LIN {X 0,Y 198.265,Z 302.232,A -85,B 0,C 180,E1 -25531.624,E2 -25531.624} C_VEL
LIN {X 0,Y 201.477,Z 266.48,A -85,B 0,C 180,E1 -25532.577,E2 -25532.577} C_VEL
LIN {X 0,Y 197.128,Z 257.364,A -85,B 0,C 180,E1 -25535.935,E2 -25535.935} C_VEL
LIN {X 0,Y 193.487,Z 250.577,A -85,B 0,C 180,E1 -25539.188,E2 -25539.188} C_VEL
LIN {X 0,Y 190.353,Z 244.979,A -85,B 0,C 180,E1 -25542.543,E2 -25542.543} C_VEL
LIN {X 0,Y 187.689,Z 240.639,A -85,B 0,C 180,E1 -25546.051,E2 -25546.051} C_VEL
LIN {X 0,Y 185.533,Z 236.807,A -85,B 0,C 180,E1 -25549.91,E2 -25549.91} C_VEL
LIN {X 0,Y 183.726,Z 233.495,A -85,B 0,C 180,E1 -25555.359,E2 -25555.359} C_VEL
LIN {X 0,Y 183.496,Z 232.327,A -85,B 0,C 180,E1 -25557.256,E2 -25557.256} C_VEL
LIN {X 0,Y 183.478,Z 232.249,A -85,B 0,C 180,E1 -25562.195,E2 -25562.195} C_VEL
LIN {X 0,Y 183.641,Z 233.069,A -85,B 0,C 180,E1 -25563.703,E2 -25563.703} C_VEL
LIN {X 0,Y 185.447,Z 236.708,A -85,B 0,C 180,E1 -25569.566,E2 -25569.566} C_VEL
LIN {X 0,Y 186.036,Z 237.651,A -85,B 0,C 180,E1 -25570.761,E2 -25570.761} C_VEL
LIN {X 0,Y 188.522,Z 241.906,A -85,B 0,C 180,E1 -25574.781,E2 -25574.781} C_VEL
LIN {X 0,Y 190.791,Z 245.771,A -85,B 0,C 180,E1 -25577.622,E2 -25577.622} C_VEL
LIN {X 0,Y 194.145,Z 251.69,A -85,B 0,C 180,E1 -25581.084,E2 -25581.084} C_VEL
LIN {X 0,Y 196.253,Z 256.423,A -85,B 0,C 180,E1 -25583.047,E2 -25583.047} C_VEL
LIN {X 0,Y 199.614,Z 265.237,A -85,B 0,C 180,E1 -25585.917,E2 -25585.917} C_VEL
LIN {X 0,Y 201.248,Z 269.943,A -85,B 0,C 180,E1 -25587.212,E2 -25587.212} C_VEL
LIN {X 0,Y 196.172,Z 324.072,A -85,B 0,C 180,E1 -25588.661,E2 -25588.661} C_VEL
LIN {X 0,Y 193.425,Z 339.856,A -85,B 0,C 180,E1 -25589.304,E2 -25589.304} C_VEL
LIN {X 0,Y 189.575,Z 355.078,A -85,B 0,C 180,E1 -25590.202,E2 -25590.202} C_VEL
LIN {X 0,Y 185.022,Z 368.797,A -85,B 0,C 180,E1 -25591.278,E2 -25591.278} C_VEL
LIN {X 0,Y 179.622,Z 382.244,A -85,B 0,C 180,E1 -25592.73,E2 -25592.73} C_VEL
LIN {X 0,Y 173.751,Z 394.633,A -85,B 0,C 180,E1 -25594.491,E2 -25594.491} C_VEL
LIN {X 0,Y 166.772,Z 407.28,A -85,B 0,C 180,E1 -25596.804,E2 -25596.804} C_VEL
LIN {X 0,Y 159.475,Z 418.758,A -85,B 0,C 180,E1 -25599.536,E2 -25599.536} C_VEL
LIN {X 0,Y 152.63,Z 428.424,A -85,B 0,C 180,E1 -25602.545,E2 -25602.545} C_VEL
LIN {X 0,Y 146.12,Z 436.937,A -85,B 0,C 180,E1 -25605.972,E2 -25605.972} C_VEL
LIN {X 0,Y 139.146,Z 445.515,A -85,B 0,C 180,E1 -25610.535,E2 -25610.535} C_VEL
LIN {X 0,Y 132.201,Z 453.257,A -85,B 0,C 180,E1 -25616.069,E2 -25616.069} C_VEL
LIN {X 0,Y 127.367,Z 458.659,A -85,B 0,C 180,E1 -25621.381,E2 -25621.381} C_VEL
LIN {X 0,Y 125.007,Z 460.662,A -85,B 0,C 180,E1 -25623.675,E2 -25623.675} C_VEL
LIN {X 0,Y 119.764,Z 463.476,A -85,B 0,C 180,E1 -25627.4,E2 -25627.4} C_VEL
LIN {X 0,Y 115.776,Z 465.338,A -85,B 0,C 180,E1 -25630.633,E2 -25630.633} C_VEL
LIN {X 0,Y 113.774,Z 466.531,A -85,B 0,C 180,E1 -25633.354,E2 -25633.354} C_VEL
LIN {X 0,Y 113.422,Z 466.832,A -85,B 0,C 180,E1 -25634.315,E2 -25634.315} C_VEL
LIN {X 0,Y 112.458,Z 468.336,A -85,B 0,C 180,E1 -25639.194,E2 -25639.194} C_VEL
LIN {X 0,Y 112.095,Z 469.523,A -85,B 0,C 180,E1 -25646.405,E2 -25646.405} C_VEL
LIN {X 0,Y 112.248,Z 469.683,A -85,B 0,C 180,E1 -25650,E2 -25650} C_VEL
LIN {X 0,Y 112.127,Z 469.052,A -85,B 0,C 180,E1 -25657.201,E2 -25657.201} C_VEL
LIN {X 0,Y 113.102,Z 467.265,A -85,B 0,C 180,E1 -25664.392,E2 -25664.392} C_VEL
LIN {X 0,Y 115.542,Z 464.307,A -85,B 0,C 180,E1 -25671.405,E2 -25671.405} C_VEL
LIN {X 0,Y 119.379,Z 460.108,A -85,B 0,C 180,E1 -25678.097,E2 -25678.097} C_VEL
LIN {X 0,Y 124.74,Z 454.565,A -85,B 0,C 180,E1 -25684.292,E2 -25684.292} C_VEL
LIN {X 0,Y 131.461,Z 447.53,A -85,B 0,C 180,E1 -25689.906,E2 -25689.906} C_VEL
LIN {X 0,Y 138.147,Z 439.961,A -85,B 0,C 180,E1 -25694.428,E2 -25694.428} C_VEL
LIN {X 0,Y 145.577,Z 430.948,A -85,B 0,C 180,E1 -25698.443,E2 -25698.443} C_VEL
LIN {X 0,Y 153.784,Z 420.066,A -85,B 0,C 180,E1 -25702.03,E2 -25702.03} C_VEL
LIN {X 0,Y 161.304,Z 408.87,A -85,B 0,C 180,E1 -25704.78,E2 -25704.78} C_VEL
LIN {X 0,Y 168.57,Z 396.421,A -85,B 0,C 180,E1 -25707.123,E2 -25707.123} C_VEL
LIN {X 0,Y 175.175,Z 383.102,A -85,B 0,C 180,E1 -25709.044,E2 -25709.044} C_VEL
LIN {X 0,Y 180.736,Z 369.84,A -85,B 0,C 180,E1 -25710.466,E2 -25710.466} C_VEL
LIN {X 0,Y 185.351,Z 356.452,A -85,B 0,C 180,E1 -25711.547,E2 -25711.547} C_VEL
LIN {X 0,Y 189.311,Z 341.786,A -85,B 0,C 180,E1 -25712.417,E2 -25712.417} C_VEL
LIN {X 0,Y 192.254,Z 326.282,A -85,B 0,C 180,E1 -25713.068,E2 -25713.068} C_VEL
LIN {X 0,Y 194.747,Z 303.203,A -85,B 0,C 180,E1 -25713.707,E2 -25713.707} C_VEL
LIN {X 0,Y 197.576,Z 272.684,A -85,B 0,C 180,E1 -25714.507,E2 -25714.507} C_VEL
LIN {X 0,Y 194.287,Z 263.272,A -85,B 0,C 180,E1 -25717.468,E2 -25717.468} C_VEL
LIN {X 0,Y 192.199,Z 258.069,A -85,B 0,C 180,E1 -25719.533,E2 -25719.533} C_VEL
LIN {X 0,Y 189.081,Z 252.283,A -85,B 0,C 180,E1 -25722.91,E2 -25722.91} C_VEL
LIN {X 0,Y 186.331,Z 247.346,A -85,B 0,C 180,E1 -25726.643,E2 -25726.643} C_VEL
LIN {X 0,Y 184.285,Z 243.616,A -85,B 0,C 180,E1 -25730.396,E2 -25730.396} C_VEL
LIN {X 0,Y 182.602,Z 240.468,A -85,B 0,C 180,E1 -25735.447,E2 -25735.447} C_VEL
LIN {X 0,Y 182.361,Z 239.282,A -85,B 0,C 180,E1 -25737.239,E2 -25737.239} C_VEL
LIN {X 0,Y 182.233,Z 239.216,A -85,B 0,C 180,E1 -25742.21,E2 -25742.21} C_VEL
LIN {X 0,Y 182.442,Z 239.623,A -85,B 0,C 180,E1 -25743.866,E2 -25743.866} C_VEL
LIN {X 0,Y 183.716,Z 242.998,A -85,B 0,C 180,E1 -25748.802,E2 -25748.802} C_VEL
LIN {X 0,Y 184.522,Z 244.089,A -85,B 0,C 180,E1 -25750.562,E2 -25750.562} C_VEL
LIN {X 0,Y 186.922,Z 248.505,A -85,B 0,C 180,E1 -25754.702,E2 -25754.702} C_VEL
LIN {X 0,Y 189.301,Z 252.766,A -85,B 0,C 180,E1 -25757.8,E2 -25757.8} C_VEL
LIN {X 0,Y 192.242,Z 258.192,A -85,B 0,C 180,E1 -25760.952,E2 -25760.952} C_VEL
LIN {X 0,Y 195.843,Z 265.523,A -85,B 0,C 180,E1 -25764.233,E2 -25764.233} C_VEL
LIN {X 0,Y 197.757,Z 269.776,A -85,B 0,C 180,E1 -25765.802,E2 -25765.802} C_VEL
LIN {X 0,Y 193.116,Z 318.432,A -85,B 0,C 180,E1 -25767.116,E2 -25767.116} C_VEL
LIN {X 0,Y 190.335,Z 334.317,A -85,B 0,C 180,E1 -25767.744,E2 -25767.744} C_VEL
LIN {X 0,Y 186.373,Z 350.163,A -85,B 0,C 180,E1 -25768.748,E2 -25768.748} C_VEL
LIN {X 0,Y 181.609,Z 364.66,A -85,B 0,C 180,E1 -25770.016,E2 -25770.016} C_VEL
LIN {X 0,Y 176.331,Z 377.734,A -85,B 0,C 180,E1 -25771.522,E2 -25771.522} C_VEL
LIN {X 0,Y 169.714,Z 391.314,A -85,B 0,C 180,E1 -25773.551,E2 -25773.551} C_VEL
LIN {X 0,Y 162.629,Z 403.514,A -85,B 0,C 180,E1 -25775.877,E2 -25775.877} C_VEL
LIN {X 0,Y 155.241,Z 414.63,A -85,B 0,C 180,E1 -25778.654,E2 -25778.654} C_VEL
LIN {X 0,Y 148.173,Z 424.142,A -85,B 0,C 180,E1 -25781.784,E2 -25781.784} C_VEL
LIN {X 0,Y 141.937,Z 431.925,A -85,B 0,C 180,E1 -25785.123,E2 -25785.123} C_VEL
LIN {X 0,Y 134.944,Z 439.778,A -85,B 0,C 180,E1 -25789.382,E2 -25789.382} C_VEL
LIN {X 0,Y 127.923,Z 447.104,A -85,B 0,C 180,E1 -25794.77,E2 -25794.77} C_VEL
LIN {X 0,Y 122.164,Z 452.906,A -85,B 0,C 180,E1 -25800.725,E2 -25800.725} C_VEL
LIN {X 0,Y 118.72,Z 456.337,A -85,B 0,C 180,E1 -25805.519,E2 -25805.519} C_VEL
LIN {X 0,Y 115.274,Z 459.803,A -85,B 0,C 180,E1 -25812.252,E2 -25812.252} C_VEL
LIN {X 0,Y 113.203,Z 462.086,A -85,B 0,C 180,E1 -25819.266,E2 -25819.266} C_VEL
LIN {X 0,Y 112.353,Z 463.242,A -85,B 0,C 180,E1 -25826.414,E2 -25826.414} C_VEL
LIN {X 0,Y 112.335,Z 463.394,A -85,B 0,C 180,E1 -25830,E2 -25830} C_VEL
LIN {X 0,Y 112.624,Z 462.835,A -85,B 0,C 180,E1 -25837.17,E2 -25837.17} C_VEL
LIN {X 0,Y 114.052,Z 461.162,A -85,B 0,C 180,E1 -25844.27,E2 -25844.27} C_VEL
LIN {X 0,Y 116.719,Z 458.337,A -85,B 0,C 180,E1 -25851.179,E2 -25851.179} C_VEL
LIN {X 0,Y 120.935,Z 454.278,A -85,B 0,C 180,E1 -25857.705,E2 -25857.705} C_VEL
LIN {X 0,Y 126.325,Z 448.897,A -85,B 0,C 180,E1 -25863.804,E2 -25863.804} C_VEL
LIN {X 0,Y 133.008,Z 442.029,A -85,B 0,C 180,E1 -25869.351,E2 -25869.351} C_VEL
LIN {X 0,Y 140.793,Z 433.449,A -85,B 0,C 180,E1 -25874.335,E2 -25874.335} C_VEL
LIN {X 0,Y 148.026,Z 424.662,A -85,B 0,C 180,E1 -25878.165,E2 -25878.165} C_VEL
LIN {X 0,Y 155.16,Z 415.03,A -85,B 0,C 180,E1 -25881.384,E2 -25881.384} C_VEL
LIN {X 0,Y 163.16,Z 402.982,A -85,B 0,C 180,E1 -25884.393,E2 -25884.393} C_VEL
LIN {X 0,Y 170.261,Z 390.675,A -85,B 0,C 180,E1 -25886.707,E2 -25886.707} C_VEL
LIN {X 0,Y 176.412,Z 378.03,A -85,B 0,C 180,E1 -25888.585,E2 -25888.585} C_VEL
LIN {X 0,Y 181.47,Z 365.506,A -85,B 0,C 180,E1 -25890.06,E2 -25890.06} C_VEL
LIN {X 0,Y 186.272,Z 351.22,A -85,B 0,C 180,E1 -25891.309,E2 -25891.309} C_VEL
LIN {X 0,Y 190.119,Z 336.499,A -85,B 0,C 180,E1 -25892.238,E2 -25892.238} C_VEL
LIN {X 0,Y 192.878,Z 321.586,A -85,B 0,C 180,E1 -25892.902,E2 -25892.902} C_VEL
LIN {X 0,Y 195.246,Z 299.869,A -85,B 0,C 180,E1 -25893.515,E2 -25893.515} C_VEL
LIN {X 0,Y 198.046,Z 270.082,A -85,B 0,C 180,E1 -25894.274,E2 -25894.274} C_VEL
LIN {X 0,Y 194.366,Z 262.13,A -85,B 0,C 180,E1 -25897.389,E2 -25897.389} C_VEL
LIN {X 0,Y 190.853,Z 255.339,A -85,B 0,C 180,E1 -25900.854,E2 -25900.854} C_VEL
LIN {X 0,Y 188.192,Z 250.581,A -85,B 0,C 180,E1 -25904.013,E2 -25904.013} C_VEL
LIN {X 0,Y 186.382,Z 247.347,A -85,B 0,C 180,E1 -25906.639,E2 -25906.639} C_VEL
LIN {X 0,Y 184.409,Z 243.664,A -85,B 0,C 180,E1 -25910.402,E2 -25910.402} C_VEL
LIN {X 0,Y 182.727,Z 240.167,A -85,B 0,C 180,E1 -25916.14,E2 -25916.14} C_VEL
LIN {X 0,Y 182.572,Z 239.291,A -85,B 0,C 180,E1 -25917.794,E2 -25917.794} C_VEL
LIN {X 0,Y 182.613,Z 239.299,A -85,B 0,C 180,E1 -25922.205,E2 -25922.205} C_VEL
LIN {X 0,Y 184.443,Z 243.691,A -85,B 0,C 180,E1 -25929.319,E2 -25929.319} C_VEL
LIN {X 0,Y 187.034,Z 248.381,A -85,B 0,C 180,E1 -25933.998,E2 -25933.998} C_VEL
LIN {X 0,Y 189.551,Z 252.95,A -85,B 0,C 180,E1 -25937.324,E2 -25937.324} C_VEL
LIN {X 0,Y 192.628,Z 258.726,A -85,B 0,C 180,E1 -25940.628,E2 -25940.628} C_VEL
LIN {X 0,Y 195.09,Z 265.052,A -85,B 0,C 180,E1 -25943.041,E2 -25943.041} C_VEL
LIN {X 0,Y 197.801,Z 272.956,A -85,B 0,C 180,E1 -25945.465,E2 -25945.465} C_VEL
LIN {X 0,Y 192.844,Z 324.07,A -85,B 0,C 180,E1 -25946.818,E2 -25946.818} C_VEL
LIN {X 0,Y 190.047,Z 339.667,A -85,B 0,C 180,E1 -25947.435,E2 -25947.435} C_VEL
LIN {X 0,Y 186.087,Z 354.885,A -85,B 0,C 180,E1 -25948.303,E2 -25948.303} C_VEL
LIN {X 0,Y 181.436,Z 368.604,A -85,B 0,C 180,E1 -25949.361,E2 -25949.361} C_VEL
LIN {X 0,Y 175.871,Z 382.05,A -85,B 0,C 180,E1 -25950.776,E2 -25950.776} C_VEL
LIN {X 0,Y 169.385,Z 395.286,A -85,B 0,C 180,E1 -25952.642,E2 -25952.642} C_VEL
LIN {X 0,Y 161.958,Z 408.156,A -85,B 0,C 180,E1 -25955.009,E2 -25955.009} C_VEL
LIN {X 0,Y 153.809,Z 420.321,A -85,B 0,C 180,E1 -25957.982,E2 -25957.982} C_VEL
LIN {X 0,Y 145.602,Z 431.152,A -85,B 0,C 180,E1 -25961.568,E2 -25961.568} C_VEL
LIN {X 0,Y 138.413,Z 439.903,A -85,B 0,C 180,E1 -25965.472,E2 -25965.472} C_VEL
LIN {X 0,Y 131.53,Z 447.689,A -85,B 0,C 180,E1 -25970.119,E2 -25970.119} C_VEL
LIN {X 0,Y 126.304,Z 453.057,A -85,B 0,C 180,E1 -25974.249,E2 -25974.249} C_VEL
LIN {X 0,Y 120.674,Z 458.941,A -85,B 0,C 180,E1 -25980.328,E2 -25980.328} C_VEL
LIN {X 0,Y 117.361,Z 462.447,A -85,B 0,C 180,E1 -25985.217,E2 -25985.217} C_VEL
LIN {X 0,Y 114.102,Z 465.992,A -85,B 0,C 180,E1 -25992.063,E2 -25992.063} C_VEL
LIN {X 0,Y 113.422,Z 466.832,A -85,B 0,C 180,E1 -25994.315,E2 -25994.315} C_VEL
LIN {X 0,Y 112.199,Z 467.828,A -85,B 0,C 180,E1 -25997.204,E2 -25997.204} C_VEL
LIN {X 0,Y 108.998,Z 468.967,A -85,B 0,C 180,E1 -26002.012,E2 -26002.012} C_VEL
LIN {X 0,Y 105.596,Z 469.509,A -85,B 0,C 180,E1 -26008.153,E2 -26008.153} C_VEL
LIN {X 0,Y 105.135,Z 469.471,A -85,B 0,C 180,E1 -26010.309,E2 -26010.309} C_VEL
LIN {X 0,Y 105.053,Z 468.852,A -85,B 0,C 180,E1 -26017.689,E2 -26017.689} C_VEL
LIN {X 0,Y 106.184,Z 467.064,A -85,B 0,C 180,E1 -26025.352,E2 -26025.352} C_VEL
LIN {X 0,Y 108.884,Z 464.105,A -85,B 0,C 180,E1 -26032.785,E2 -26032.785} C_VEL
LIN {X 0,Y 113.108,Z 459.907,A -85,B 0,C 180,E1 -26039.807,E2 -26039.807} C_VEL
LIN {X 0,Y 118.877,Z 454.363,A -85,B 0,C 180,E1 -26046.242,E2 -26046.242} C_VEL
LIN {X 0,Y 126.045,Z 447.327,A -85,B 0,C 180,E1 -26051.997,E2 -26051.997} C_VEL
LIN {X 0,Y 133.556,Z 439.265,A -85,B 0,C 180,E1 -26056.836,E2 -26056.836} C_VEL
LIN {X 0,Y 140.943,Z 430.746,A -85,B 0,C 180,E1 -26060.615,E2 -26060.615} C_VEL
LIN {X 0,Y 149.492,Z 419.863,A -85,B 0,C 180,E1 -26064.191,E2 -26064.191} C_VEL
LIN {X 0,Y 157.306,Z 408.668,A -85,B 0,C 180,E1 -26066.898,E2 -26066.898} C_VEL
LIN {X 0,Y 165.108,Z 395.702,A -85,B 0,C 180,E1 -26069.284,E2 -26069.284} C_VEL
LIN {X 0,Y 171.628,Z 382.898,A -85,B 0,C 180,E1 -26071.079,E2 -26071.079} C_VEL
LIN {X 0,Y 177.342,Z 369.636,A -85,B 0,C 180,E1 -26072.464,E2 -26072.464} C_VEL
LIN {X 0,Y 182.076,Z 356.247,A -85,B 0,C 180,E1 -26073.512,E2 -26073.512} C_VEL
LIN {X 0,Y 186.132,Z 341.578,A -85,B 0,C 180,E1 -26074.353,E2 -26074.353} C_VEL
LIN {X 0,Y 189.091,Z 326.379,A -85,B 0,C 180,E1 -26074.978,E2 -26074.978} C_VEL
LIN {X 0,Y 191.547,Z 304.546,A -85,B 0,C 180,E1 -26075.576,E2 -26075.576} C_VEL
LIN {X 0,Y 194.298,Z 275.812,A -85,B 0,C 180,E1 -26076.313,E2 -26076.313} C_VEL
LIN {X 0,Y 191.694,Z 267.952,A -85,B 0,C 180,E1 -26078.915,E2 -26078.915} C_VEL
LIN {X 0,Y 190.099,Z 263.817,A -85,B 0,C 180,E1 -26080.636,E2 -26080.636} C_VEL
LIN {X 0,Y 186.9,Z 257.529,A -85,B 0,C 180,E1 -26084.46,E2 -26084.46} C_VEL
LIN {X 0,Y 184.856,Z 253.826,A -85,B 0,C 180,E1 -26087.512,E2 -26087.512} C_VEL
LIN {X 0,Y 183.132,Z 250.42,A -85,B 0,C 180,E1 -26090.961,E2 -26090.961} C_VEL
LIN {X 0,Y 181.628,Z 247.298,A -85,B 0,C 180,E1 -26095.979,E2 -26095.979} C_VEL
LIN {X 0,Y 181.494,Z 246.355,A -85,B 0,C 180,E1 -26097.226,E2 -26097.226} C_VEL
LIN {X 0,Y 181.279,Z 246.096,A -85,B 0,C 180,E1 -26100,E2 -26100} C_VEL
LIN {X 0,Y 181.526,Z 246.656,A -85,B 0,C 180,E1 -26103.607,E2 -26103.607} C_VEL
LIN {X 0,Y 182.764,Z 250.033,A -85,B 0,C 180,E1 -26108.639,E2 -26108.639} C_VEL
LIN {X 0,Y 183.445,Z 251.083,A -85,B 0,C 180,E1 -26110.206,E2 -26110.206} C_VEL
LIN {X 0,Y 185.533,Z 255.12,A -85,B 0,C 180,E1 -26114.029,E2 -26114.029} C_VEL
LIN {X 0,Y 187.886,Z 259.548,A -85,B 0,C 180,E1 -26117.272,E2 -26117.272} C_VEL
LIN {X 0,Y 190.91,Z 265.585,A -85,B 0,C 180,E1 -26120.664,E2 -26120.664} C_VEL
LIN {X 0,Y 193.676,Z 271.568,A -85,B 0,C 180,E1 -26123.317,E2 -26123.317} C_VEL
LIN {X 0,Y 194.461,Z 273.393,A -85,B 0,C 180,E1 -26124.018,E2 -26124.018} C_VEL
LIN {X 0,Y 189.897,Z 319.326,A -85,B 0,C 180,E1 -26125.238,E2 -26125.238} C_VEL
LIN {X 0,Y 187.147,Z 334.525,A -85,B 0,C 180,E1 -26125.828,E2 -26125.828} C_VEL
LIN {X 0,Y 183.063,Z 350.369,A -85,B 0,C 180,E1 -26126.799,E2 -26126.799} C_VEL
LIN {X 0,Y 178.165,Z 364.865,A -85,B 0,C 180,E1 -26128.04,E2 -26128.04} C_VEL
LIN {X 0,Y 172.564,Z 378.281,A -85,B 0,C 180,E1 -26129.56,E2 -26129.56} C_VEL
LIN {X 0,Y 165.9,Z 391.516,A -85,B 0,C 180,E1 -26131.509,E2 -26131.509} C_VEL
LIN {X 0,Y 158.581,Z 403.716,A -85,B 0,C 180,E1 -26133.802,E2 -26133.802} C_VEL
LIN {X 0,Y 150.896,Z 414.832,A -85,B 0,C 180,E1 -26136.542,E2 -26136.542} C_VEL
LIN {X 0,Y 143.09,Z 424.887,A -85,B 0,C 180,E1 -26139.858,E2 -26139.858} C_VEL
LIN {X 0,Y 136.996,Z 432.126,A -85,B 0,C 180,E1 -26143.027,E2 -26143.027} C_VEL
LIN {X 0,Y 129.619,Z 439.979,A -85,B 0,C 180,E1 -26147.331,E2 -26147.331} C_VEL
LIN {X 0,Y 122.176,Z 447.304,A -85,B 0,C 180,E1 -26152.843,E2 -26152.843} C_VEL
LIN {X 0,Y 115.98,Z 453.107,A -85,B 0,C 180,E1 -26158.998,E2 -26158.998} C_VEL
LIN {X 0,Y 112.283,Z 456.537,A -85,B 0,C 180,E1 -26164.015,E2 -26164.015} C_VEL
LIN {X 0,Y 108.496,Z 460.004,A -85,B 0,C 180,E1 -26171.102,E2 -26171.102} C_VEL
LIN {X 0,Y 106.216,Z 462.286,A -85,B 0,C 180,E1 -26178.551,E2 -26178.551} C_VEL
LIN {X 0,Y 105.265,Z 463.441,A -85,B 0,C 180,E1 -26186.172,E2 -26186.172} C_VEL
LIN {X 0,Y 105.237,Z 463.593,A -85,B 0,C 180,E1 -26190,E2 -26190} C_VEL
LIN {X 0,Y 105.593,Z 463.033,A -85,B 0,C 180,E1 -26197.65,E2 -26197.65} C_VEL
LIN {X 0,Y 107.158,Z 461.361,A -85,B 0,C 180,E1 -26205.209,E2 -26205.209} C_VEL
LIN {X 0,Y 110.095,Z 458.536,A -85,B 0,C 180,E1 -26212.521,E2 -26212.521} C_VEL
LIN {X 0,Y 114.638,Z 454.478,A -85,B 0,C 180,E1 -26219.37,E2 -26219.37} C_VEL
LIN {X 0,Y 120.451,Z 449.095,A -85,B 0,C 180,E1 -26225.696,E2 -26225.696} C_VEL
LIN {X 0,Y 127.581,Z 442.227,A -85,B 0,C 180,E1 -26231.38,E2 -26231.38} C_VEL
LIN {X 0,Y 134.691,Z 434.842,A -85,B 0,C 180,E1 -26235.845,E2 -26235.845} C_VEL
LIN {X 0,Y 141.616,Z 426.984,A -85,B 0,C 180,E1 -26239.422,E2 -26239.422} C_VEL
LIN {X 0,Y 148.352,Z 418.465,A -85,B 0,C 180,E1 -26242.516,E2 -26242.516} C_VEL
LIN {X 0,Y 155.929,Z 408.058,A -85,B 0,C 180,E1 -26245.343,E2 -26245.343} C_VEL
LIN {X 0,Y 163.074,Z 396.737,A -85,B 0,C 180,E1 -26247.756,E2 -26247.756} C_VEL
LIN {X 0,Y 169.836,Z 384.428,A -85,B 0,C 180,E1 -26249.75,E2 -26249.75} C_VEL
LIN {X 0,Y 175.956,Z 370.966,A -85,B 0,C 180,E1 -26251.489,E2 -26251.489} C_VEL
LIN {X 0,Y 181.231,Z 356.999,A -85,B 0,C 180,E1 -26252.811,E2 -26252.811} C_VEL
LIN {X 0,Y 185.502,Z 342.638,A -85,B 0,C 180,E1 -26253.824,E2 -26253.824} C_VEL
LIN {X 0,Y 188.751,Z 327.83,A -85,B 0,C 180,E1 -26254.581,E2 -26254.581} C_VEL
LIN {X 0,Y 190.91,Z 312.871,A -85,B 0,C 180,E1 -26255.085,E2 -26255.085} C_VEL
LIN {X 0,Y 194.716,Z 273.628,A -85,B 0,C 180,E1 -26256.087,E2 -26256.087} C_VEL
LIN {X 0,Y 191.419,Z 266.286,A -85,B 0,C 180,E1 -26259.194,E2 -26259.194} C_VEL
LIN {X 0,Y 188.424,Z 260.334,A -85,B 0,C 180,E1 -26262.499,E2 -26262.499} C_VEL
LIN {X 0,Y 186.354,Z 256.478,A -85,B 0,C 180,E1 -26265.238,E2 -26265.238} C_VEL
LIN {X 0,Y 185.084,Z 254.064,A -85,B 0,C 180,E1 -26267.249,E2 -26267.249} C_VEL
LIN {X 0,Y 183.296,Z 250.539,A -85,B 0,C 180,E1 -26270.899,E2 -26270.899} C_VEL
LIN {X 0,Y 181.769,Z 246.756,A -85,B 0,C 180,E1 -26276.952,E2 -26276.952} C_VEL
LIN {X 0,Y 181.705,Z 246.353,A -85,B 0,C 180,E1 -26277.783,E2 -26277.783} C_VEL
LIN {X 0,Y 181.743,Z 246.395,A -85,B 0,C 180,E1 -26282.216,E2 -26282.216} C_VEL
LIN {X 0,Y 183.21,Z 250.417,A -85,B 0,C 180,E1 -26288.548,E2 -26288.548} C_VEL
LIN {X 0,Y 183.796,Z 251.506,A -85,B 0,C 180,E1 -26289.908,E2 -26289.908} C_VEL
LIN {X 0,Y 185.704,Z 255.116,A -85,B 0,C 180,E1 -26293.403,E2 -26293.403} C_VEL
LIN {X 0,Y 188.056,Z 259.604,A -85,B 0,C 180,E1 -26296.696,E2 -26296.696} C_VEL
LIN {X 0,Y 190.88,Z 265.244,A -85,B 0,C 180,E1 -26299.912,E2 -26299.912} C_VEL
LIN {X 0,Y 193.413,Z 272.592,A -85,B 0,C 180,E1 -26302.574,E2 -26302.574} C_VEL
LIN {X 0,Y 194.513,Z 275.967,A -85,B 0,C 180,E1 -26303.639,E2 -26303.639} C_VEL
LIN {X 0,Y 189.713,Z 324.05,A -85,B 0,C 180,E1 -26304.905,E2 -26304.905} C_VEL
LIN {X 0,Y 186.883,Z 339.478,A -85,B 0,C 180,E1 -26305.503,E2 -26305.503} C_VEL
LIN {X 0,Y 182.824,Z 354.693,A -85,B 0,C 180,E1 -26306.341,E2 -26306.341} C_VEL
LIN {X 0,Y 178.063,Z 368.412,A -85,B 0,C 180,E1 -26307.369,E2 -26307.369} C_VEL
LIN {X 0,Y 172.329,Z 381.855,A -85,B 0,C 180,E1 -26308.738,E2 -26308.738} C_VEL
LIN {X 0,Y 165.946,Z 394.557,A -85,B 0,C 180,E1 -26310.492,E2 -26310.492} C_VEL
LIN {X 0,Y 158.655,Z 406.888,A -85,B 0,C 180,E1 -26312.685,E2 -26312.685} C_VEL
LIN {X 0,Y 150.774,Z 418.363,A -85,B 0,C 180,E1 -26315.34,E2 -26315.34} C_VEL
LIN {X 0,Y 143.339,Z 428.028,A -85,B 0,C 180,E1 -26318.326,E2 -26318.326} C_VEL
LIN {X 0,Y 135.276,Z 437.531,A -85,B 0,C 180,E1 -26322.24,E2 -26322.24} C_VEL
LIN {X 0,Y 128.065,Z 445.458,A -85,B 0,C 180,E1 -26326.687,E2 -26326.687} C_VEL
LIN {X 0,Y 120.559,Z 452.858,A -85,B 0,C 180,E1 -26332.258,E2 -26332.258} C_VEL
LIN {X 0,Y 114.487,Z 458.741,A -85,B 0,C 180,E1 -26338.547,E2 -26338.547} C_VEL
LIN {X 0,Y 110.903,Z 462.248,A -85,B 0,C 180,E1 -26343.666,E2 -26343.666} C_VEL
LIN {X 0,Y 107.319,Z 465.792,A -85,B 0,C 180,E1 -26350.887,E2 -26350.887} C_VEL
LIN {X 0,Y 105.463,Z 468.137,A -85,B 0,C 180,E1 -26358.468,E2 -26358.468} C_VEL
LIN {X 0,Y 105.005,Z 469.324,A -85,B 0,C 180,E1 -26366.162,E2 -26366.162} C_VEL
LIN {X 0,Y 105.135,Z 469.471,A -85,B 0,C 180,E1 -26370.309,E2 -26370.309} C_VEL
LIN {X 0,Y 104.271,Z 469.315,A -85,B 0,C 180,E1 -26373.503,E2 -26373.503} C_VEL
LIN {X 0,Y 101.54,Z 468.641,A -85,B 0,C 180,E1 -26378.803,E2 -26378.803} C_VEL
LIN {X 0,Y 99.689,Z 467.734,A -85,B 0,C 180,E1 -26383.209,E2 -26383.209} C_VEL
LIN {X 0,Y 99.403,Z 466.819,A -85,B 0,C 180,E1 -26386.595,E2 -26386.595} C_VEL
LIN {X 0,Y 99.635,Z 466.446,A -85,B 0,C 180,E1 -26387.713,E2 -26387.713} C_VEL
LIN {X 0,Y 102.3,Z 463.903,A -85,B 0,C 180,E1 -26394.343,E2 -26394.343} C_VEL
LIN {X 0,Y 106.942,Z 459.705,A -85,B 0,C 180,E1 -26401.718,E2 -26401.718} C_VEL
LIN {X 0,Y 113.158,Z 454.161,A -85,B 0,C 180,E1 -26408.395,E2 -26408.395} C_VEL
LIN {X 0,Y 120.825,Z 447.126,A -85,B 0,C 180,E1 -26414.267,E2 -26414.267} C_VEL
LIN {X 0,Y 128.169,Z 439.682,A -85,B 0,C 180,E1 -26418.852,E2 -26418.852} C_VEL
LIN {X 0,Y 136.511,Z 430.543,A -85,B 0,C 180,E1 -26422.938,E2 -26422.938} C_VEL
LIN {X 0,Y 145.416,Z 419.66,A -85,B 0,C 180,E1 -26426.481,E2 -26426.481} C_VEL
LIN {X 0,Y 154.229,Z 407.43,A -85,B 0,C 180,E1 -26429.329,E2 -26429.329} C_VEL
LIN {X 0,Y 161.72,Z 395.216,A -85,B 0,C 180,E1 -26431.513,E2 -26431.513} C_VEL
LIN {X 0,Y 168.293,Z 382.694,A -85,B 0,C 180,E1 -26433.206,E2 -26433.206} C_VEL
LIN {X 0,Y 174.176,Z 369.432,A -85,B 0,C 180,E1 -26434.533,E2 -26434.533} C_VEL
LIN {X 0,Y 179.02,Z 356.041,A -85,B 0,C 180,E1 -26435.547,E2 -26435.547} C_VEL
LIN {X 0,Y 183.161,Z 341.369,A -85,B 0,C 180,E1 -26436.362,E2 -26436.362} C_VEL
LIN {X 0,Y 186.241,Z 325.951,A -85,B 0,C 180,E1 -26436.96,E2 -26436.96} C_VEL
LIN {X 0,Y 188.908,Z 302.588,A -85,B 0,C 180,E1 -26437.572,E2 -26437.572} C_VEL
LIN {X 0,Y 191.218,Z 278.961,A -85,B 0,C 180,E1 -26438.178,E2 -26438.178} C_VEL
LIN {X 0,Y 188.79,Z 271.325,A -85,B 0,C 180,E1 -26440.92,E2 -26440.92} C_VEL
LIN {X 0,Y 186.376,Z 266.079,A -85,B 0,C 180,E1 -26443.853,E2 -26443.853} C_VEL
LIN {X 0,Y 183.976,Z 261.169,A -85,B 0,C 180,E1 -26447.452,E2 -26447.452} C_VEL
LIN {X 0,Y 182.055,Z 257.306,A -85,B 0,C 180,E1 -26451.397,E2 -26451.397} C_VEL
LIN {X 0,Y 180.654,Z 254.028,A -85,B 0,C 180,E1 -26456.655,E2 -26456.655} C_VEL
LIN {X 0,Y 180.559,Z 253.298,A -85,B 0,C 180,E1 -26457.77,E2 -26457.77} C_VEL
LIN {X 0,Y 180.502,Z 253.322,A -85,B 0,C 180,E1 -26462.232,E2 -26462.232} C_VEL
LIN {X 0,Y 180.623,Z 253.821,A -85,B 0,C 180,E1 -26463.486,E2 -26463.486} C_VEL
LIN {X 0,Y 181.897,Z 257.182,A -85,B 0,C 180,E1 -26468.681,E2 -26468.681} C_VEL
LIN {X 0,Y 182.428,Z 258.249,A -85,B 0,C 180,E1 -26469.984,E2 -26469.984} C_VEL
LIN {X 0,Y 184.187,Z 261.777,A -85,B 0,C 180,E1 -26473.375,E2 -26473.375} C_VEL
LIN {X 0,Y 186.111,Z 265.61,A -85,B 0,C 180,E1 -26476.241,E2 -26476.241} C_VEL
LIN {X 0,Y 188.905,Z 271.487,A -85,B 0,C 180,E1 -26479.637,E2 -26479.637} C_VEL
LIN {X 0,Y 191.338,Z 277.056,A -85,B 0,C 180,E1 -26482.163,E2 -26482.163} C_VEL
LIN {X 0,Y 186.913,Z 319.966,A -85,B 0,C 180,E1 -26483.286,E2 -26483.286} C_VEL
LIN {X 0,Y 184.172,Z 334.734,A -85,B 0,C 180,E1 -26483.844,E2 -26483.844} C_VEL
LIN {X 0,Y 179.971,Z 350.575,A -85,B 0,C 180,E1 -26484.779,E2 -26484.779} C_VEL
LIN {X 0,Y 174.939,Z 365.069,A -85,B 0,C 180,E1 -26485.987,E2 -26485.987} C_VEL
LIN {X 0,Y 168.998,Z 378.848,A -85,B 0,C 180,E1 -26487.518,E2 -26487.518} C_VEL
LIN {X 0,Y 162.298,Z 391.719,A -85,B 0,C 180,E1 -26489.37,E2 -26489.37} C_VEL
LIN {X 0,Y 154.746,Z 403.918,A -85,B 0,C 180,E1 -26491.618,E2 -26491.618} C_VEL
LIN {X 0,Y 146.774,Z 415.033,A -85,B 0,C 180,E1 -26494.311,E2 -26494.311} C_VEL
LIN {X 0,Y 138.223,Z 425.571,A -85,B 0,C 180,E1 -26497.778,E2 -26497.778} C_VEL
LIN {X 0,Y 131.073,Z 433.55,A -85,B 0,C 180,E1 -26501.352,E2 -26501.352} C_VEL
LIN {X 0,Y 123.433,Z 441.18,A -85,B 0,C 180,E1 -26505.774,E2 -26505.774} C_VEL
LIN {X 0,Y 116.565,Z 447.506,A -85,B 0,C 180,E1 -26510.723,E2 -26510.723} C_VEL
LIN {X 0,Y 109.923,Z 453.308,A -85,B 0,C 180,E1 -26517.081,E2 -26517.081} C_VEL
LIN {X 0,Y 105.917,Z 456.737,A -85,B 0,C 180,E1 -26522.324,E2 -26522.324} C_VEL
LIN {X 0,Y 101.776,Z 460.204,A -85,B 0,C 180,E1 -26529.802,E2 -26529.802} C_VEL
LIN {X 0,Y 99.262,Z 462.485,A -85,B 0,C 180,E1 -26537.737,E2 -26537.737} C_VEL
LIN {X 0,Y 98.189,Z 463.64,A -85,B 0,C 180,E1 -26545.896,E2 -26545.896} C_VEL
LIN {X 0,Y 98.151,Z 463.791,A -85,B 0,C 180,E1 -26550,E2 -26550} C_VEL
LIN {X 0,Y 98.553,Z 463.232,A -85,B 0,C 180,E1 -26558.2,E2 -26558.2} C_VEL
LIN {X 0,Y 100.308,Z 461.56,A -85,B 0,C 180,E1 -26566.276,E2 -26566.276} C_VEL
LIN {X 0,Y 103.541,Z 458.735,A -85,B 0,C 180,E1 -26574.033,E2 -26574.033} C_VEL
LIN {X 0,Y 108.454,Z 454.678,A -85,B 0,C 180,E1 -26581.226,E2 -26581.226} C_VEL
LIN {X 0,Y 114.73,Z 449.294,A -85,B 0,C 180,E1 -26587.776,E2 -26587.776} C_VEL
LIN {X 0,Y 122.322,Z 442.424,A -85,B 0,C 180,E1 -26593.588,E2 -26593.588} C_VEL
LIN {X 0,Y 129.836,Z 435.039,A -85,B 0,C 180,E1 -26598.098,E2 -26598.098} C_VEL
LIN {X 0,Y 138.086,Z 426.022,A -85,B 0,C 180,E1 -26602.178,E2 -26602.178} C_VEL
LIN {X 0,Y 145.406,Z 417.042,A -85,B 0,C 180,E1 -26605.253,E2 -26605.253} C_VEL
LIN {X 0,Y 153.298,Z 406.312,A -85,B 0,C 180,E1 -26608.01,E2 -26608.01} C_VEL
LIN {X 0,Y 160.782,Z 394.593,A -85,B 0,C 180,E1 -26610.316,E2 -26610.316} C_VEL
LIN {X 0,Y 167.758,Z 381.819,A -85,B 0,C 180,E1 -26612.239,E2 -26612.239} C_VEL
LIN {X 0,Y 173.403,Z 369.413,A -85,B 0,C 180,E1 -26613.731,E2 -26613.731} C_VEL
LIN {X 0,Y 178.819,Z 354.984,A -85,B 0,C 180,E1 -26615.014,E2 -26615.014} C_VEL
LIN {X 0,Y 183.041,Z 340.679,A -85,B 0,C 180,E1 -26615.938,E2 -26615.938} C_VEL
LIN {X 0,Y 186.152,Z 326.326,A -85,B 0,C 180,E1 -26616.616,E2 -26616.616} C_VEL
LIN {X 0,Y 188.281,Z 311.061,A -85,B 0,C 180,E1 -26617.085,E2 -26617.085} C_VEL
LIN {X 0,Y 191.601,Z 277.358,A -85,B 0,C 180,E1 -26617.932,E2 -26617.932} C_VEL
LIN {X 0,Y 188.939,Z 271.235,A -85,B 0,C 180,E1 -26620.723,E2 -26620.723} C_VEL
LIN {X 0,Y 186.434,Z 265.996,A -85,B 0,C 180,E1 -26623.788,E2 -26623.788} C_VEL
LIN {X 0,Y 184.009,Z 261.064,A -85,B 0,C 180,E1 -26627.524,E2 -26627.524} C_VEL
LIN {X 0,Y 182.199,Z 257.396,A -85,B 0,C 180,E1 -26631.403,E2 -26631.403} C_VEL
LIN {X 0,Y 180.838,Z 253.419,A -85,B 0,C 180,E1 -26637.772,E2 -26637.772} C_VEL
LIN {X 0,Y 180.846,Z 253.423,A -85,B 0,C 180,E1 -26641.948,E2 -26641.948} C_VEL
LIN {X 0,Y 182.229,Z 257.409,A -85,B 0,C 180,E1 -26648.315,E2 -26648.315} C_VEL
LIN {X 0,Y 184.319,Z 261.658,A -85,B 0,C 180,E1 -26652.664,E2 -26652.664} C_VEL
LIN {X 0,Y 186.661,Z 266.383,A -85,B 0,C 180,E1 -26656.155,E2 -26656.155} C_VEL
LIN {X 0,Y 189.039,Z 271.573,A -85,B 0,C 180,E1 -26659.054,E2 -26659.054} C_VEL
LIN {X 0,Y 191.237,Z 278.518,A -85,B 0,C 180,E1 -26661.561,E2 -26661.561} C_VEL
LIN {X 0,Y 191.418,Z 279.082,A -85,B 0,C 180,E1 -26661.752,E2 -26661.752} C_VEL
LIN {X 0,Y 187.991,Z 314.374,A -85,B 0,C 180,E1 -26662.676,E2 -26662.676} C_VEL
LIN {X 0,Y 185.758,Z 330.481,A -85,B 0,C 180,E1 -26663.153,E2 -26663.153} C_VEL
LIN {X 0,Y 182.418,Z 345.389,A -85,B 0,C 180,E1 -26663.791,E2 -26663.791} C_VEL
LIN {X 0,Y 177.908,Z 360.157,A -85,B 0,C 180,E1 -26664.689,E2 -26664.689} C_VEL
LIN {X 0,Y 172.683,Z 373.545,A -85,B 0,C 180,E1 -26665.78,E2 -26665.78} C_VEL
LIN {X 0,Y 166.858,Z 386.011,A -85,B 0,C 180,E1 -26667.154,E2 -26667.154} C_VEL
LIN {X 0,Y 159.505,Z 399.343,A -85,B 0,C 180,E1 -26669.108,E2 -26669.108} C_VEL
LIN {X 0,Y 152.155,Z 410.729,A -85,B 0,C 180,E1 -26671.294,E2 -26671.294} C_VEL
LIN {X 0,Y 144.133,Z 421.561,A -85,B 0,C 180,E1 -26674.011,E2 -26674.011} C_VEL
LIN {X 0,Y 135.297,Z 432.117,A -85,B 0,C 180,E1 -26677.611,E2 -26677.611} C_VEL
LIN {X 0,Y 127.517,Z 440.582,A -85,B 0,C 180,E1 -26681.575,E2 -26681.575} C_VEL
LIN {X 0,Y 120.864,Z 447.29,A -85,B 0,C 180,E1 -26685.751,E2 -26685.751} C_VEL
LIN {X 0,Y 113.201,Z 454.285,A -85,B 0,C 180,E1 -26691.622,E2 -26691.622} C_VEL
LIN {X 0,Y 106.329,Z 460.444,A -85,B 0,C 180,E1 -26699.232,E2 -26699.232} C_VEL
LIN {X 0,Y 102.354,Z 463.975,A -85,B 0,C 180,E1 -26705.67,E2 -26705.67} C_VEL
LIN {X 0,Y 99.3,Z 466.911,A -85,B 0,C 180,E1 -26713.554,E2 -26713.554} C_VEL
LIN {X 0,Y 98.006,Z 468.673,A -85,B 0,C 180,E1 -26721.754,E2 -26721.754} C_VEL
LIN {X 0,Y 98.071,Z 469.286,A -85,B 0,C 180,E1 -26730,E2 -26730} C_VEL
LIN {X 0,Y 98.004,Z 468.653,A -85,B 0,C 180,E1 -26738.246,E2 -26738.246} C_VEL
LIN {X 0,Y 99.285,Z 466.863,A -85,B 0,C 180,E1 -26746.448,E2 -26746.448} C_VEL
LIN {X 0,Y 99.635,Z 466.446,A -85,B 0,C 180,E1 -26747.713,E2 -26747.713} C_VEL
LIN {X 0,Y 100.092,Z 465.362,A -85,B 0,C 180,E1 -26751.029,E2 -26751.029} C_VEL
LIN {X 0,Y 99.735,Z 463.166,A -85,B 0,C 180,E1 -26756.581,E2 -26756.581} C_VEL
LIN {X 0,Y 99.944,Z 461.097,A -85,B 0,C 180,E1 -26760.993,E2 -26760.993} C_VEL
LIN {X 0,Y 101.224,Z 459.313,A -85,B 0,C 180,E1 -26764.125,E2 -26764.125} C_VEL
LIN {X 0,Y 101.962,Z 458.648,A -85,B 0,C 180,E1 -26765.091,E2 -26765.091} C_VEL
LIN {X 0,Y 109.528,Z 452.329,A -85,B 0,C 180,E1 -26772.357,E2 -26772.357} C_VEL
LIN {X 0,Y 117.944,Z 444.89,A -85,B 0,C 180,E1 -26778.146,E2 -26778.146} C_VEL
LIN {X 0,Y 126.039,Z 436.932,A -85,B 0,C 180,E1 -26782.616,E2 -26782.616} C_VEL
LIN {X 0,Y 134.924,Z 427.394,A -85,B 0,C 180,E1 -26786.451,E2 -26786.451} C_VEL
LIN {X 0,Y 142.961,Z 417.679,A -85,B 0,C 180,E1 -26789.351,E2 -26789.351} C_VEL
LIN {X 0,Y 151.42,Z 406.154,A -85,B 0,C 180,E1 -26791.869,E2 -26791.869} C_VEL
LIN {X 0,Y 158.593,Z 394.751,A -85,B 0,C 180,E1 -26793.815,E2 -26793.815} C_VEL
LIN {X 0,Y 165.199,Z 382.49,A -85,B 0,C 180,E1 -26795.416,E2 -26795.416} C_VEL
LIN {X 0,Y 171.242,Z 369.227,A -85,B 0,C 180,E1 -26796.679,E2 -26796.679} C_VEL
LIN {X 0,Y 176.58,Z 354.705,A -85,B 0,C 180,E1 -26797.724,E2 -26797.724} C_VEL
LIN {X 0,Y 180.816,Z 339.634,A -85,B 0,C 180,E1 -26798.499,E2 -26798.499} C_VEL
LIN {X 0,Y 183.883,Z 323.989,A -85,B 0,C 180,E1 -26799.045,E2 -26799.045} C_VEL
LIN {X 0,Y 188.346,Z 282.194,A -85,B 0,C 180,E1 -26800.094,E2 -26800.094} C_VEL
LIN {X 0,Y 186.475,Z 276.204,A -85,B 0,C 180,E1 -26802.452,E2 -26802.452} C_VEL
LIN {X 0,Y 183.982,Z 270.588,A -85,B 0,C 180,E1 -26805.906,E2 -26805.906} C_VEL
LIN {X 0,Y 182.185,Z 266.965,A -85,B 0,C 180,E1 -26809.02,E2 -26809.02} C_VEL
LIN {X 0,Y 180.959,Z 264.175,A -85,B 0,C 180,E1 -26811.907,E2 -26811.907} C_VEL
LIN {X 0,Y 179.688,Z 260.55,A -85,B 0,C 180,E1 -26817.619,E2 -26817.619} C_VEL
LIN {X 0,Y 179.561,Z 260.263,A -85,B 0,C 180,E1 -26821.122,E2 -26821.122} C_VEL
LIN {X 0,Y 179.713,Z 260.853,A -85,B 0,C 180,E1 -26823.223,E2 -26823.223} C_VEL
LIN {X 0,Y 180.946,Z 264.221,A -85,B 0,C 180,E1 -26828.516,E2 -26828.516} C_VEL
LIN {X 0,Y 182.835,Z 268.358,A -85,B 0,C 180,E1 -26832.656,E2 -26832.656} C_VEL
LIN {X 0,Y 184.578,Z 272.076,A -85,B 0,C 180,E1 -26835.458,E2 -26835.458} C_VEL
LIN {X 0,Y 187.357,Z 278.295,A -85,B 0,C 180,E1 -26839.055,E2 -26839.055} C_VEL
LIN {X 0,Y 188.408,Z 280.84,A -85,B 0,C 180,E1 -26840.25,E2 -26840.25} C_VEL
LIN {X 0,Y 184.341,Z 319.511,A -85,B 0,C 180,E1 -26841.243,E2 -26841.243} C_VEL
LIN {X 0,Y 181.608,Z 334.089,A -85,B 0,C 180,E1 -26841.756,E2 -26841.756} C_VEL
LIN {X 0,Y 177.493,Z 349.631,A -85,B 0,C 180,E1 -26842.619,E2 -26842.619} C_VEL
LIN {X 0,Y 172.677,Z 363.418,A -85,B 0,C 180,E1 -26843.686,E2 -26843.686} C_VEL
LIN {X 0,Y 166.424,Z 377.855,A -85,B 0,C 180,E1 -26845.191,E2 -26845.191} C_VEL
LIN {X 0,Y 158.933,Z 391.921,A -85,B 0,C 180,E1 -26847.136,E2 -26847.136} C_VEL
LIN {X 0,Y 151.142,Z 404.12,A -85,B 0,C 180,E1 -26849.324,E2 -26849.324} C_VEL
LIN {X 0,Y 142.896,Z 415.235,A -85,B 0,C 180,E1 -26851.962,E2 -26851.962} C_VEL
LIN {X 0,Y 134.568,Z 425.038,A -85,B 0,C 180,E1 -26855.064,E2 -26855.064} C_VEL
LIN {X 0,Y 126.495,Z 433.751,A -85,B 0,C 180,E1 -26858.937,E2 -26858.937} C_VEL
LIN {X 0,Y 118.418,Z 441.382,A -85,B 0,C 180,E1 -26863.362,E2 -26863.362} C_VEL
LIN {X 0,Y 111.147,Z 447.706,A -85,B 0,C 180,E1 -26868.4,E2 -26868.4} C_VEL
LIN {X 0,Y 104.007,Z 453.509,A -85,B 0,C 180,E1 -26874.945,E2 -26874.945} C_VEL
LIN {X 0,Y 99.646,Z 456.938,A -85,B 0,C 180,E1 -26880.415,E2 -26880.415} C_VEL
LIN {X 0,Y 95.123,Z 460.404,A -85,B 0,C 180,E1 -26888.321,E2 -26888.321} C_VEL
LIN {X 0,Y 92.315,Z 462.685,A -85,B 0,C 180,E1 -26896.798,E2 -26896.798} C_VEL
LIN {X 0,Y 91.106,Z 463.839,A -85,B 0,C 180,E1 -26905.576,E2 -26905.576} C_VEL
LIN {X 0,Y 91.056,Z 463.99,A -85,B 0,C 180,E1 -26910,E2 -26910} C_VEL
LIN {X 0,Y 91.542,Z 463.43,A -85,B 0,C 180,E1 -26918.833,E2 -26918.833} C_VEL
LIN {X 0,Y 93.476,Z 461.76,A -85,B 0,C 180,E1 -26927.502,E2 -26927.502} C_VEL
LIN {X 0,Y 97.067,Z 458.934,A -85,B 0,C 180,E1 -26935.749,E2 -26935.749} C_VEL
LIN {X 0,Y 102.403,Z 454.877,A -85,B 0,C 180,E1 -26943.302,E2 -26943.302} C_VEL
LIN {X 0,Y 109.176,Z 449.492,A -85,B 0,C 180,E1 -26950.071,E2 -26950.071} C_VEL
LIN {X 0,Y 117.248,Z 442.623,A -85,B 0,C 180,E1 -26955.997,E2 -26955.997} C_VEL
LIN {X 0,Y 125.205,Z 435.236,A -85,B 0,C 180,E1 -26960.518,E2 -26960.518} C_VEL
LIN {X 0,Y 133.364,Z 426.715,A -85,B 0,C 180,E1 -26964.393,E2 -26964.393} C_VEL
LIN {X 0,Y 141.464,Z 417.239,A -85,B 0,C 180,E1 -26967.626,E2 -26967.626} C_VEL
LIN {X 0,Y 149.647,Z 406.508,A -85,B 0,C 180,E1 -26970.324,E2 -26970.324} C_VEL
LIN {X 0,Y 157.389,Z 394.788,A -85,B 0,C 180,E1 -26972.56,E2 -26972.56} C_VEL
LIN {X 0,Y 164.409,Z 382.322,A -85,B 0,C 180,E1 -26974.391,E2 -26974.391} C_VEL
LIN {X 0,Y 170.382,Z 369.606,A -85,B 0,C 180,E1 -26975.871,E2 -26975.871} C_VEL
LIN {X 0,Y 175.948,Z 355.174,A -85,B 0,C 180,E1 -26977.103,E2 -26977.103} C_VEL
LIN {X 0,Y 180.257,Z 340.868,A -85,B 0,C 180,E1 -26978.004,E2 -26978.004} C_VEL
LIN {X 0,Y 183.525,Z 326.112,A -85,B 0,C 180,E1 -26978.658,E2 -26978.658} C_VEL
LIN {X 0,Y 185.726,Z 310.411,A -85,B 0,C 180,E1 -26979.115,E2 -26979.115} C_VEL
LIN {X 0,Y 188.677,Z 281.074,A -85,B 0,C 180,E1 -26979.851,E2 -26979.851} C_VEL
LIN {X 0,Y 186.061,Z 274.979,A -85,B 0,C 180,E1 -26982.978,E2 -26982.978} C_VEL
LIN {X 0,Y 183.778,Z 270.029,A -85,B 0,C 180,E1 -26986.302,E2 -26986.302} C_VEL
LIN {X 0,Y 182.357,Z 267.075,A -85,B 0,C 180,E1 -26988.889,E2 -26988.889} C_VEL
LIN {X 0,Y 181.143,Z 264.284,A -85,B 0,C 180,E1 -26991.845,E2 -26991.845} C_VEL
LIN {X 0,Y 179.926,Z 260.412,A -85,B 0,C 180,E1 -26998.321,E2 -26998.321} C_VEL
LIN {X 0,Y 179.949,Z 260.479,A -85,B 0,C 180,E1 -27001.678,E2 -27001.678} C_VEL
LIN {X 0,Y 181.451,Z 264.902,A -85,B 0,C 180,E1 -27008.632,E2 -27008.632} C_VEL
LIN {X 0,Y 183.183,Z 268.723,A -85,B 0,C 180,E1 -27012.322,E2 -27012.322} C_VEL
LIN {X 0,Y 185.331,Z 273.268,A -85,B 0,C 180,E1 -27015.675,E2 -27015.675} C_VEL
LIN {X 0,Y 187.142,Z 277.578,A -85,B 0,C 180,E1 -27018.048,E2 -27018.048} C_VEL
LIN {X 0,Y 188.59,Z 282.469,A -85,B 0,C 180,E1 -27019.88,E2 -27019.88} C_VEL
LIN {X 0,Y 184.279,Z 323.036,A -85,B 0,C 180,E1 -27020.869,E2 -27020.869} C_VEL
LIN {X 0,Y 181.223,Z 339.099,A -85,B 0,C 180,E1 -27021.449,E2 -27021.449} C_VEL
LIN {X 0,Y 176.983,Z 354.31,A -85,B 0,C 180,E1 -27022.219,E2 -27022.219} C_VEL
LIN {X 0,Y 171.983,Z 368.025,A -85,B 0,C 180,E1 -27023.153,E2 -27023.153} C_VEL
LIN {X 0,Y 165.957,Z 381.466,A -85,B 0,C 180,E1 -27024.426,E2 -27024.426} C_VEL
LIN {X 0,Y 158.625,Z 395.161,A -85,B 0,C 180,E1 -27026.208,E2 -27026.208} C_VEL
LIN {X 0,Y 150.715,Z 407.567,A -85,B 0,C 180,E1 -27028.337,E2 -27028.337} C_VEL
LIN {X 0,Y 141.621,Z 419.728,A -85,B 0,C 180,E1 -27031.125,E2 -27031.125} C_VEL
LIN {X 0,Y 132.343,Z 430.558,A -85,B 0,C 180,E1 -27034.601,E2 -27034.601} C_VEL
LIN {X 0,Y 124.87,Z 438.372,A -85,B 0,C 180,E1 -27038.004,E2 -27038.004} C_VEL
LIN {X 0,Y 115.845,Z 447.091,A -85,B 0,C 180,E1 -27043.28,E2 -27043.28} C_VEL
LIN {X 0,Y 107.669,Z 454.086,A -85,B 0,C 180,E1 -27049.251,E2 -27049.251} C_VEL
LIN {X 0,Y 100.977,Z 459.598,A -85,B 0,C 180,E1 -27056.165,E2 -27056.165} C_VEL
LIN {X 0,Y 95.859,Z 463.775,A -85,B 0,C 180,E1 -27063.902,E2 -27063.902} C_VEL
LIN {X 0,Y 92.447,Z 466.711,A -85,B 0,C 180,E1 -27072.296,E2 -27072.296} C_VEL
LIN {X 0,Y 90.951,Z 468.474,A -85,B 0,C 180,E1 -27081.109,E2 -27081.109} C_VEL
LIN {X 0,Y 90.969,Z 469.087,A -85,B 0,C 180,E1 -27090,E2 -27090} C_VEL
LIN {X 0,Y 90.95,Z 468.453,A -85,B 0,C 180,E1 -27098.89,E2 -27098.89} C_VEL
LIN {X 0,Y 92.651,Z 466.429,A -85,B 0,C 180,E1 -27108.461,E2 -27108.461} C_VEL
LIN {X 0,Y 95.801,Z 463.701,A -85,B 0,C 180,E1 -27116.114,E2 -27116.114} C_VEL
LIN {X 0,Y 100.912,Z 459.503,A -85,B 0,C 180,E1 -27123.859,E2 -27123.859} C_VEL
LIN {X 0,Y 101.962,Z 458.648,A -85,B 0,C 180,E1 -27125.091,E2 -27125.091} C_VEL
LIN {X 0,Y 103.958,Z 456.64,A -85,B 0,C 180,E1 -27127.969,E2 -27127.969} C_VEL
LIN {X 0,Y 106.169,Z 453.069,A -85,B 0,C 180,E1 -27132.857,E2 -27132.857} C_VEL
LIN {X 0,Y 108.888,Z 449.011,A -85,B 0,C 180,E1 -27137.457,E2 -27137.457} C_VEL
LIN {X 0,Y 111.565,Z 446.226,A -85,B 0,C 180,E1 -27139.784,E2 -27139.784} C_VEL
LIN {X 0,Y 120.56,Z 437.969,A -85,B 0,C 180,E1 -27144.699,E2 -27144.699} C_VEL
LIN {X 0,Y 129.744,Z 428.684,A -85,B 0,C 180,E1 -27148.556,E2 -27148.556} C_VEL
LIN {X 0,Y 138.044,Z 419.255,A -85,B 0,C 180,E1 -27151.428,E2 -27151.428} C_VEL
LIN {X 0,Y 147.467,Z 407.024,A -85,B 0,C 180,E1 -27154.099,E2 -27154.099} C_VEL
LIN {X 0,Y 155.58,Z 394.548,A -85,B 0,C 180,E1 -27156.171,E2 -27156.171} C_VEL
LIN {X 0,Y 162.367,Z 382.286,A -85,B 0,C 180,E1 -27157.7,E2 -27157.7} C_VEL
LIN {X 0,Y 168.554,Z 369.023,A -85,B 0,C 180,E1 -27158.899,E2 -27158.899} C_VEL
LIN {X 0,Y 174.01,Z 354.499,A -85,B 0,C 180,E1 -27159.89,E2 -27159.89} C_VEL
LIN {X 0,Y 178.335,Z 339.426,A -85,B 0,C 180,E1 -27160.623,E2 -27160.623} C_VEL
LIN {X 0,Y 181.423,Z 324,A -85,B 0,C 180,E1 -27161.136,E2 -27161.136} C_VEL
LIN {X 0,Y 185.65,Z 285.548,A -85,B 0,C 180,E1 -27162.09,E2 -27162.09} C_VEL
LIN {X 0,Y 184.57,Z 281.992,A -85,B 0,C 180,E1 -27163.611,E2 -27163.611} C_VEL
LIN {X 0,Y 182.399,Z 276.822,A -85,B 0,C 180,E1 -27166.917,E2 -27166.917} C_VEL
LIN {X 0,Y 180.896,Z 273.547,A -85,B 0,C 180,E1 -27169.79,E2 -27169.79} C_VEL
LIN {X 0,Y 179.88,Z 271.026,A -85,B 0,C 180,E1 -27172.423,E2 -27172.423} C_VEL
LIN {X 0,Y 178.762,Z 267.395,A -85,B 0,C 180,E1 -27178.311,E2 -27178.311} C_VEL
LIN {X 0,Y 178.696,Z 267.303,A -85,B 0,C 180,E1 -27181.127,E2 -27181.127} C_VEL
LIN {X 0,Y 178.802,Z 267.759,A -85,B 0,C 180,E1 -27182.816,E2 -27182.816} C_VEL
LIN {X 0,Y 179.82,Z 270.978,A -85,B 0,C 180,E1 -27187.863,E2 -27187.863} C_VEL
LIN {X 0,Y 181.595,Z 275.146,A -85,B 0,C 180,E1 -27192.09,E2 -27192.09} C_VEL
LIN {X 0,Y 183.304,Z 278.985,A -85,B 0,C 180,E1 -27194.999,E2 -27194.999} C_VEL
LIN {X 0,Y 185.694,Z 284.816,A -85,B 0,C 180,E1 -27198.301,E2 -27198.301} C_VEL
LIN {X 0,Y 181.791,Z 320.368,A -85,B 0,C 180,E1 -27199.187,E2 -27199.187} C_VEL
LIN {X 0,Y 179.102,Z 334.3,A -85,B 0,C 180,E1 -27199.65,E2 -27199.65} C_VEL
LIN {X 0,Y 174.894,Z 349.837,A -85,B 0,C 180,E1 -27200.479,E2 -27200.479} C_VEL
LIN {X 0,Y 169.956,Z 363.623,A -85,B 0,C 180,E1 -27201.5,E2 -27201.5} C_VEL
LIN {X 0,Y 163.278,Z 378.569,A -85,B 0,C 180,E1 -27203,E2 -27203} C_VEL
LIN {X 0,Y 155.828,Z 392.124,A -85,B 0,C 180,E1 -27204.816,E2 -27204.816} C_VEL
LIN {X 0,Y 147.793,Z 404.322,A -85,B 0,C 180,E1 -27206.922,E2 -27206.922} C_VEL
LIN {X 0,Y 139.259,Z 415.437,A -85,B 0,C 180,E1 -27209.476,E2 -27209.476} C_VEL
LIN {X 0,Y 130.195,Z 425.699,A -85,B 0,C 180,E1 -27212.671,E2 -27212.671} C_VEL
LIN {X 0,Y 122.157,Z 433.952,A -85,B 0,C 180,E1 -27216.346,E2 -27216.346} C_VEL
LIN {X 0,Y 113.646,Z 441.583,A -85,B 0,C 180,E1 -27220.751,E2 -27220.751} C_VEL
LIN {X 0,Y 105.925,Z 447.907,A -85,B 0,C 180,E1 -27225.84,E2 -27225.84} C_VEL
LIN {X 0,Y 98.251,Z 453.709,A -85,B 0,C 180,E1 -27232.554,E2 -27232.554} C_VEL
LIN {X 0,Y 93.505,Z 457.139,A -85,B 0,C 180,E1 -27238.256,E2 -27238.256} C_VEL
LIN {X 0,Y 88.53,Z 460.605,A -85,B 0,C 180,E1 -27246.614,E2 -27246.614} C_VEL
LIN {X 0,Y 85.411,Z 462.884,A -85,B 0,C 180,E1 -27255.709,E2 -27255.709} C_VEL
LIN {X 0,Y 84.05,Z 464.037,A -85,B 0,C 180,E1 -27265.204,E2 -27265.204} C_VEL
LIN {X 0,Y 83.956,Z 464.189,A -85,B 0,C 180,E1 -27270,E2 -27270} C_VEL
LIN {X 0,Y 84.514,Z 463.629,A -85,B 0,C 180,E1 -27279.574,E2 -27279.574} C_VEL
LIN {X 0,Y 86.704,Z 461.959,A -85,B 0,C 180,E1 -27288.919,E2 -27288.919} C_VEL
LIN {X 0,Y 90.694,Z 459.133,A -85,B 0,C 180,E1 -27297.707,E2 -27297.707} C_VEL
LIN {X 0,Y 96.509,Z 455.076,A -85,B 0,C 180,E1 -27305.632,E2 -27305.632} C_VEL
LIN {X 0,Y 103.811,Z 449.691,A -85,B 0,C 180,E1 -27312.61,E2 -27312.61} C_VEL
LIN {X 0,Y 112.409,Z 442.821,A -85,B 0,C 180,E1 -27318.613,E2 -27318.613} C_VEL
LIN {X 0,Y 120.812,Z 435.433,A -85,B 0,C 180,E1 -27323.119,E2 -27323.119} C_VEL
LIN {X 0,Y 128.924,Z 427.346,A -85,B 0,C 180,E1 -27326.786,E2 -27326.786} C_VEL
LIN {X 0,Y 137.793,Z 417.435,A -85,B 0,C 180,E1 -27330.12,E2 -27330.12} C_VEL
LIN {X 0,Y 146.258,Z 406.704,A -85,B 0,C 180,E1 -27332.744,E2 -27332.744} C_VEL
LIN {X 0,Y 154.241,Z 394.984,A -85,B 0,C 180,E1 -27334.905,E2 -27334.905} C_VEL
LIN {X 0,Y 160.906,Z 383.598,A -85,B 0,C 180,E1 -27336.526,E2 -27336.526} C_VEL
LIN {X 0,Y 166.849,Z 371.546,A -85,B 0,C 180,E1 -27337.925,E2 -27337.925} C_VEL
LIN {X 0,Y 172.544,Z 357.575,A -85,B 0,C 180,E1 -27339.113,E2 -27339.113} C_VEL
LIN {X 0,Y 177.154,Z 343.208,A -85,B 0,C 180,E1 -27340.006,E2 -27340.006} C_VEL
LIN {X 0,Y 180.846,Z 327.483,A -85,B 0,C 180,E1 -27340.712,E2 -27340.712} C_VEL
LIN {X 0,Y 183.153,Z 312.058,A -85,B 0,C 180,E1 -27341.159,E2 -27341.159} C_VEL
LIN {X 0,Y 185.941,Z 284.998,A -85,B 0,C 180,E1 -27341.83,E2 -27341.83} C_VEL
LIN {X 0,Y 183.718,Z 279.618,A -85,B 0,C 180,E1 -27344.883,E2 -27344.883} C_VEL
LIN {X 0,Y 181.876,Z 275.393,A -85,B 0,C 180,E1 -27348.012,E2 -27348.012} C_VEL
LIN {X 0,Y 180.05,Z 271.097,A -85,B 0,C 180,E1 -27352.43,E2 -27352.43} C_VEL
LIN {X 0,Y 179.061,Z 267.452,A -85,B 0,C 180,E1 -27358.313,E2 -27358.313} C_VEL
LIN {X 0,Y 179.062,Z 267.596,A -85,B 0,C 180,E1 -27361.546,E2 -27361.546} C_VEL
LIN {X 0,Y 180.359,Z 271.739,A -85,B 0,C 180,E1 -27368.12,E2 -27368.12} C_VEL
LIN {X 0,Y 181.967,Z 275.553,A -85,B 0,C 180,E1 -27371.805,E2 -27371.805} C_VEL
LIN {X 0,Y 183.891,Z 279.968,A -85,B 0,C 180,E1 -27375.02,E2 -27375.02} C_VEL
LIN {X 0,Y 185.351,Z 283.728,A -85,B 0,C 180,E1 -27377.089,E2 -27377.089} C_VEL
LIN {X 0,Y 185.907,Z 285.784,A -85,B 0,C 180,E1 -27377.885,E2 -27377.885} C_VEL
LIN {X 0,Y 181.765,Z 323.512,A -85,B 0,C 180,E1 -27378.8,E2 -27378.8} C_VEL
LIN {X 0,Y 178.745,Z 338.91,A -85,B 0,C 180,E1 -27379.326,E2 -27379.326} C_VEL
LIN {X 0,Y 174.418,Z 354.118,A -85,B 0,C 180,E1 -27380.055,E2 -27380.055} C_VEL
LIN {X 0,Y 169.314,Z 367.832,A -85,B 0,C 180,E1 -27380.941,E2 -27380.941} C_VEL
LIN {X 0,Y 163.145,Z 381.272,A -85,B 0,C 180,E1 -27382.152,E2 -27382.152} C_VEL
LIN {X 0,Y 156.348,Z 393.673,A -85,B 0,C 180,E1 -27383.669,E2 -27383.669} C_VEL
LIN {X 0,Y 149.296,Z 404.725,A -85,B 0,C 180,E1 -27385.438,E2 -27385.438} C_VEL
LIN {X 0,Y 140.919,Z 415.983,A -85,B 0,C 180,E1 -27387.718,E2 -27387.718} C_VEL
LIN {X 0,Y 132.495,Z 425.943,A -85,B 0,C 180,E1 -27390.462,E2 -27390.462} C_VEL
LIN {X 0,Y 123.135,Z 435.695,A -85,B 0,C 180,E1 -27394.147,E2 -27394.147} C_VEL
LIN {X 0,Y 114.505,Z 443.843,A -85,B 0,C 180,E1 -27398.504,E2 -27398.504} C_VEL
LIN {X 0,Y 106.519,Z 450.586,A -85,B 0,C 180,E1 -27403.467,E2 -27403.467} C_VEL
LIN {X 0,Y 98.541,Z 456.817,A -85,B 0,C 180,E1 -27410.067,E2 -27410.067} C_VEL
LIN {X 0,Y 92.082,Z 461.647,A -85,B 0,C 180,E1 -27417.706,E2 -27417.706} C_VEL
LIN {X 0,Y 87.321,Z 465.193,A -85,B 0,C 180,E1 -27426.27,E2 -27426.27} C_VEL
LIN {X 0,Y 84.558,Z 467.537,A -85,B 0,C 180,E1 -27435.561,E2 -27435.561} C_VEL
LIN {X 0,Y 83.728,Z 468.727,A -85,B 0,C 180,E1 -27445.185,E2 -27445.185} C_VEL
LIN {X 0,Y 83.875,Z 468.888,A -85,B 0,C 180,E1 -27450,E2 -27450} C_VEL
LIN {X 0,Y 83.728,Z 468.72,A -85,B 0,C 180,E1 -27454.815,E2 -27454.815} C_VEL
LIN {X 0,Y 84.552,Z 467.501,A -85,B 0,C 180,E1 -27464.44,E2 -27464.44} C_VEL
LIN {X 0,Y 87.29,Z 465.13,A -85,B 0,C 180,E1 -27473.738,E2 -27473.738} C_VEL
LIN {X 0,Y 91.987,Z 461.56,A -85,B 0,C 180,E1 -27482.331,E2 -27482.331} C_VEL
LIN {X 0,Y 98.494,Z 456.706,A -85,B 0,C 180,E1 -27489.955,E2 -27489.955} C_VEL
LIN {X 0,Y 106.482,Z 450.436,A -85,B 0,C 180,E1 -27496.554,E2 -27496.554} C_VEL
LIN {X 0,Y 111.565,Z 446.226,A -85,B 0,C 180,E1 -27499.784,E2 -27499.784} C_VEL
LIN {X 0,Y 114.352,Z 443.364,A -85,B 0,C 180,E1 -27501.983,E2 -27501.983} C_VEL
LIN {X 0,Y 121.01,Z 434.264,A -85,B 0,C 180,E1 -27508.741,E2 -27508.741} C_VEL
LIN {X 0,Y 123.952,Z 430.797,A -85,B 0,C 180,E1 -27510.495,E2 -27510.495} C_VEL
LIN {X 0,Y 125.106,Z 429.569,A -85,B 0,C 180,E1 -27510.959,E2 -27510.959} C_VEL
LIN {X 0,Y 134.77,Z 419.052,A -85,B 0,C 180,E1 -27514.1,E2 -27514.1} C_VEL
LIN {X 0,Y 144.484,Z 406.82,A -85,B 0,C 180,E1 -27516.653,E2 -27516.653} C_VEL
LIN {X 0,Y 152.839,Z 394.344,A -85,B 0,C 180,E1 -27518.616,E2 -27518.616} C_VEL
LIN {X 0,Y 159.81,Z 382.083,A -85,B 0,C 180,E1 -27520.054,E2 -27520.054} C_VEL
LIN {X 0,Y 166.127,Z 368.818,A -85,B 0,C 180,E1 -27521.187,E2 -27521.187} C_VEL
LIN {X 0,Y 171.303,Z 355.423,A -85,B 0,C 180,E1 -27522.047,E2 -27522.047} C_VEL
LIN {X 0,Y 175.708,Z 340.744,A -85,B 0,C 180,E1 -27522.738,E2 -27522.738} C_VEL
LIN {X 0,Y 178.952,Z 325.501,A -85,B 0,C 180,E1 -27523.238,E2 -27523.238} C_VEL
LIN {X 0,Y 181.721,Z 303.11,A -85,B 0,C 180,E1 -27523.764,E2 -27523.764} C_VEL
LIN {X 0,Y 183.197,Z 289.154,A -85,B 0,C 180,E1 -27524.096,E2 -27524.096} C_VEL
LIN {X 0,Y 181.554,Z 284.746,A -85,B 0,C 180,E1 -27526.712,E2 -27526.712} C_VEL
LIN {X 0,Y 179.886,Z 280.597,A -85,B 0,C 180,E1 -27530.016,E2 -27530.016} C_VEL
LIN {X 0,Y 178.79,Z 277.855,A -85,B 0,C 180,E1 -27533.015,E2 -27533.015} C_VEL
LIN {X 0,Y 177.891,Z 274.494,A -85,B 0,C 180,E1 -27538.302,E2 -27538.302} C_VEL
LIN {X 0,Y 177.861,Z 274.406,A -85,B 0,C 180,E1 -27541.698,E2 -27541.698} C_VEL
LIN {X 0,Y 179.024,Z 278.512,A -85,B 0,C 180,E1 -27548.182,E2 -27548.182} C_VEL
LIN {X 0,Y 180.439,Z 282.074,A -85,B 0,C 180,E1 -27551.65,E2 -27551.65} C_VEL
LIN {X 0,Y 182.075,Z 286.078,A -85,B 0,C 180,E1 -27554.602,E2 -27554.602} C_VEL
LIN {X 0,Y 183.152,Z 288.903,A -85,B 0,C 180,E1 -27556.259,E2 -27556.259} C_VEL
LIN {X 0,Y 179.558,Z 320.755,A -85,B 0,C 180,E1 -27557.058,E2 -27557.058} C_VEL
LIN {X 0,Y 176.651,Z 335.36,A -85,B 0,C 180,E1 -27557.524,E2 -27557.524} C_VEL
LIN {X 0,Y 172.151,Z 351.192,A -85,B 0,C 180,E1 -27558.345,E2 -27558.345} C_VEL
LIN {X 0,Y 166.704,Z 365.683,A -85,B 0,C 180,E1 -27559.387,E2 -27559.387} C_VEL
LIN {X 0,Y 160.358,Z 379.29,A -85,B 0,C 180,E1 -27560.724,E2 -27560.724} C_VEL
LIN {X 0,Y 152.988,Z 392.326,A -85,B 0,C 180,E1 -27562.406,E2 -27562.406} C_VEL
LIN {X 0,Y 144.713,Z 404.524,A -85,B 0,C 180,E1 -27564.412,E2 -27564.412} C_VEL
LIN {X 0,Y 135.906,Z 415.638,A -85,B 0,C 180,E1 -27566.87,E2 -27566.87} C_VEL
LIN {X 0,Y 126.081,Z 426.322,A -85,B 0,C 180,E1 -27570.111,E2 -27570.111} C_VEL
LIN {X 0,Y 116.742,Z 435.368,A -85,B 0,C 180,E1 -27574.13,E2 -27574.13} C_VEL
LIN {X 0,Y 107.901,Z 442.784,A -85,B 0,C 180,E1 -27578.592,E2 -27578.592} C_VEL
LIN {X 0,Y 98.738,Z 449.707,A -85,B 0,C 180,E1 -27584.62,E2 -27584.62} C_VEL
LIN {X 0,Y 90.842,Z 455.137,A -85,B 0,C 180,E1 -27591.763,E2 -27591.763} C_VEL
LIN {X 0,Y 84.489,Z 459.227,A -85,B 0,C 180,E1 -27600.06,E2 -27600.06} C_VEL
LIN {X 0,Y 80.054,Z 462.087,A -85,B 0,C 180,E1 -27609.442,E2 -27609.442} C_VEL
LIN {X 0,Y 77.513,Z 463.798,A -85,B 0,C 180,E1 -27619.553,E2 -27619.553} C_VEL
LIN {X 0,Y 76.883,Z 464.387,A -85,B 0,C 180,E1 -27630,E2 -27630} C_VEL
LIN {X 0,Y 77.511,Z 463.828,A -85,B 0,C 180,E1 -27640.448,E2 -27640.448} C_VEL
LIN {X 0,Y 80.003,Z 462.158,A -85,B 0,C 180,E1 -27650.572,E2 -27650.572} C_VEL
LIN {X 0,Y 84.447,Z 459.332,A -85,B 0,C 180,E1 -27659.957,E2 -27659.957} C_VEL
LIN {X 0,Y 90.802,Z 455.275,A -85,B 0,C 180,E1 -27668.258,E2 -27668.258} C_VEL
LIN {X 0,Y 98.675,Z 449.89,A -85,B 0,C 180,E1 -27675.418,E2 -27675.418} C_VEL
LIN {X 0,Y 107.829,Z 443.019,A -85,B 0,C 180,E1 -27681.456,E2 -27681.456} C_VEL
LIN {X 0,Y 116.682,Z 435.63,A -85,B 0,C 180,E1 -27685.914,E2 -27685.914} C_VEL
LIN {X 0,Y 124.667,Z 428.029,A -85,B 0,C 180,E1 -27689.33,E2 -27689.33} C_VEL
LIN {X 0,Y 132.96,Z 419.251,A -85,B 0,C 180,E1 -27692.298,E2 -27692.298} C_VEL
LIN {X 0,Y 141.669,Z 408.844,A -85,B 0,C 180,E1 -27694.872,E2 -27694.872} C_VEL
LIN {X 0,Y 149.862,Z 397.517,A -85,B 0,C 180,E1 -27696.977,E2 -27696.977} C_VEL
LIN {X 0,Y 157.45,Z 385.206,A -85,B 0,C 180,E1 -27698.715,E2 -27698.715} C_VEL
LIN {X 0,Y 164.312,Z 371.739,A -85,B 0,C 180,E1 -27700.22,E2 -27700.22} C_VEL
LIN {X 0,Y 170.149,Z 357.767,A -85,B 0,C 180,E1 -27701.341,E2 -27701.341} C_VEL
LIN {X 0,Y 174.856,Z 343.398,A -85,B 0,C 180,E1 -27702.191,E2 -27702.191} C_VEL
LIN {X 0,Y 178.608,Z 327.76,A -85,B 0,C 180,E1 -27702.859,E2 -27702.859} C_VEL
LIN {X 0,Y 180.9,Z 312.872,A -85,B 0,C 180,E1 -27703.275,E2 -27703.275} C_VEL
LIN {X 0,Y 183.412,Z 289.059,A -85,B 0,C 180,E1 -27703.87,E2 -27703.87} C_VEL
LIN {X 0,Y 181.298,Z 283.682,A -85,B 0,C 180,E1 -27707.334,E2 -27707.334} C_VEL
LIN {X 0,Y 179.838,Z 280.227,A -85,B 0,C 180,E1 -27710.439,E2 -27710.439} C_VEL
LIN {X 0,Y 178.997,Z 277.945,A -85,B 0,C 180,E1 -27712.952,E2 -27712.952} C_VEL
LIN {X 0,Y 178.163,Z 274.462,A -85,B 0,C 180,E1 -27718.87,E2 -27718.87} C_VEL
LIN {X 0,Y 178.175,Z 274.536,A -85,B 0,C 180,E1 -27721.13,E2 -27721.13} C_VEL
LIN {X 0,Y 179.321,Z 278.72,A -85,B 0,C 180,E1 -27727.734,E2 -27727.734} C_VEL
LIN {X 0,Y 180.798,Z 282.48,A -85,B 0,C 180,E1 -27731.349,E2 -27731.349} C_VEL
LIN {X 0,Y 182.478,Z 286.65,A -85,B 0,C 180,E1 -27734.355,E2 -27734.355} C_VEL
LIN {X 0,Y 183.46,Z 289.377,A -85,B 0,C 180,E1 -27735.877,E2 -27735.877} C_VEL
LIN {X 0,Y 179.627,Z 323.178,A -85,B 0,C 180,E1 -27736.65,E2 -27736.65} C_VEL
LIN {X 0,Y 176.524,Z 338.72,A -85,B 0,C 180,E1 -27737.152,E2 -27737.152} C_VEL
LIN {X 0,Y 172.109,Z 353.926,A -85,B 0,C 180,E1 -27737.832,E2 -27737.832} C_VEL
LIN {X 0,Y 166.911,Z 367.639,A -85,B 0,C 180,E1 -27738.666,E2 -27738.666} C_VEL
LIN {X 0,Y 160.595,Z 381.078,A -85,B 0,C 180,E1 -27739.797,E2 -27739.797} C_VEL
LIN {X 0,Y 153.627,Z 393.478,A -85,B 0,C 180,E1 -27741.235,E2 -27741.235} C_VEL
LIN {X 0,Y 146.227,Z 404.734,A -85,B 0,C 180,E1 -27742.948,E2 -27742.948} C_VEL
LIN {X 0,Y 137.749,Z 415.786,A -85,B 0,C 180,E1 -27745.093,E2 -27745.093} C_VEL
LIN {X 0,Y 129.025,Z 425.745,A -85,B 0,C 180,E1 -27747.731,E2 -27747.731} C_VEL
LIN {X 0,Y 119.254,Z 435.495,A -85,B 0,C 180,E1 -27751.291,E2 -27751.291} C_VEL
LIN {X 0,Y 110.192,Z 443.644,A -85,B 0,C 180,E1 -27755.59,E2 -27755.59} C_VEL
LIN {X 0,Y 101.735,Z 450.387,A -85,B 0,C 180,E1 -27760.544,E2 -27760.544} C_VEL
LIN {X 0,Y 93.136,Z 456.617,A -85,B 0,C 180,E1 -27767.223,E2 -27767.223} C_VEL
LIN {X 0,Y 86.093,Z 461.446,A -85,B 0,C 180,E1 -27775.15,E2 -27775.15} C_VEL
LIN {X 0,Y 80.812,Z 464.993,A -85,B 0,C 180,E1 -27784.225,E2 -27784.225} C_VEL
LIN {X 0,Y 77.637,Z 467.337,A -85,B 0,C 180,E1 -27794.242,E2 -27794.242} C_VEL
LIN {X 0,Y 76.621,Z 468.527,A -85,B 0,C 180,E1 -27804.737,E2 -27804.737} C_VEL
LIN {X 0,Y 76.771,Z 468.69,A -85,B 0,C 180,E1 -27810,E2 -27810} C_VEL
LIN {X 0,Y 76.878,Z 468.053,A -85,B 0,C 180,E1 -27820.535,E2 -27820.535} C_VEL
LIN {X 0,Y 78.896,Z 466.259,A -85,B 0,C 180,E1 -27830.874,E2 -27830.874} C_VEL
LIN {X 0,Y 83.15,Z 463.298,A -85,B 0,C 180,E1 -27840.473,E2 -27840.473} C_VEL
LIN {X 0,Y 89.348,Z 459.099,A -85,B 0,C 180,E1 -27848.996,E2 -27848.996} C_VEL
LIN {X 0,Y 97.218,Z 453.554,A -85,B 0,C 180,E1 -27856.295,E2 -27856.295} C_VEL
LIN {X 0,Y 106.486,Z 446.519,A -85,B 0,C 180,E1 -27862.372,E2 -27862.372} C_VEL
LIN {X 0,Y 115.351,Z 438.908,A -85,B 0,C 180,E1 -27867.02,E2 -27867.02} C_VEL
LIN {X 0,Y 125.106,Z 429.569,A -85,B 0,C 180,E1 -27870.959,E2 -27870.959} C_VEL
LIN {X 0,Y 128.328,Z 425.888,A -85,B 0,C 180,E1 -27872.426,E2 -27872.426} C_VEL
LIN {X 0,Y 136.035,Z 414.506,A -85,B 0,C 180,E1 -27877.354,E2 -27877.354} C_VEL
LIN {X 0,Y 139,Z 410.305,A -85,B 0,C 180,E1 -27878.588,E2 -27878.588} C_VEL
LIN {X 0,Y 140.113,Z 408.837,A -85,B 0,C 180,E1 -27878.895,E2 -27878.895} C_VEL
LIN {X 0,Y 148.807,Z 396.556,A -85,B 0,C 180,E1 -27880.836,E2 -27880.836} C_VEL
LIN {X 0,Y 156.722,Z 383.31,A -85,B 0,C 180,E1 -27882.351,E2 -27882.351} C_VEL
LIN {X 0,Y 163.155,Z 370.381,A -85,B 0,C 180,E1 -27883.423,E2 -27883.423} C_VEL
LIN {X 0,Y 168.842,Z 356.346,A -85,B 0,C 180,E1 -27884.276,E2 -27884.276} C_VEL
LIN {X 0,Y 173.53,Z 341.298,A -85,B 0,C 180,E1 -27884.946,E2 -27884.946} C_VEL
LIN {X 0,Y 176.917,Z 325.962,A -85,B 0,C 180,E1 -27885.419,E2 -27885.419} C_VEL
LIN {X 0,Y 179.621,Z 305.024,A -85,B 0,C 180,E1 -27885.902,E2 -27885.902} C_VEL
LIN {X 0,Y 180.893,Z 293.293,A -85,B 0,C 180,E1 -27886.172,E2 -27886.172} C_VEL
LIN {X 0,Y 179.286,Z 288.907,A -85,B 0,C 180,E1 -27889.269,E2 -27889.269} C_VEL
LIN {X 0,Y 177.853,Z 284.869,A -85,B 0,C 180,E1 -27893.192,E2 -27893.192} C_VEL
LIN {X 0,Y 176.989,Z 281.431,A -85,B 0,C 180,E1 -27898.863,E2 -27898.863} C_VEL
LIN {X 0,Y 176.991,Z 281.495,A -85,B 0,C 180,E1 -27901.707,E2 -27901.707} C_VEL
LIN {X 0,Y 177.956,Z 285.356,A -85,B 0,C 180,E1 -27907.66,E2 -27907.66} C_VEL
LIN {X 0,Y 179.272,Z 288.975,A -85,B 0,C 180,E1 -27911.161,E2 -27911.161} C_VEL
LIN {X 0,Y 180.732,Z 292.881,A -85,B 0,C 180,E1 -27913.995,E2 -27913.995} C_VEL
LIN {X 0,Y 180.841,Z 293.198,A -85,B 0,C 180,E1 -27914.186,E2 -27914.186} C_VEL
LIN {X 0,Y 177.582,Z 321.104,A -85,B 0,C 180,E1 -27914.873,E2 -27914.873} C_VEL
LIN {X 0,Y 174.651,Z 335.568,A -85,B 0,C 180,E1 -27915.31,E2 -27915.31} C_VEL
LIN {X 0,Y 170.049,Z 351.398,A -85,B 0,C 180,E1 -27916.074,E2 -27916.074} C_VEL
LIN {X 0,Y 164.487,Z 365.887,A -85,B 0,C 180,E1 -27917.056,E2 -27917.056} C_VEL
LIN {X 0,Y 158.197,Z 379.095,A -85,B 0,C 180,E1 -27918.265,E2 -27918.265} C_VEL
LIN {X 0,Y 150.429,Z 392.528,A -85,B 0,C 180,E1 -27919.909,E2 -27919.909} C_VEL
LIN {X 0,Y 141.912,Z 404.727,A -85,B 0,C 180,E1 -27921.787,E2 -27921.787} C_VEL
LIN {X 0,Y 132.847,Z 415.84,A -85,B 0,C 180,E1 -27924.136,E2 -27924.136} C_VEL
LIN {X 0,Y 123.789,Z 425.401,A -85,B 0,C 180,E1 -27926.862,E2 -27926.862} C_VEL
LIN {X 0,Y 114.305,Z 434.354,A -85,B 0,C 180,E1 -27930.595,E2 -27930.595} C_VEL
LIN {X 0,Y 104.899,Z 441.985,A -85,B 0,C 180,E1 -27934.843,E2 -27934.843} C_VEL
LIN {X 0,Y 96.205,Z 448.309,A -85,B 0,C 180,E1 -27939.91,E2 -27939.91} C_VEL
LIN {X 0,Y 88.113,Z 453.646,A -85,B 0,C 180,E1 -27946.124,E2 -27946.124} C_VEL
LIN {X 0,Y 81.721,Z 457.54,A -85,B 0,C 180,E1 -27952.987,E2 -27952.987} C_VEL
LIN {X 0,Y 75.638,Z 461.006,A -85,B 0,C 180,E1 -27962.317,E2 -27962.317} C_VEL
LIN {X 0,Y 71.703,Z 463.283,A -85,B 0,C 180,E1 -27972.9,E2 -27972.9} C_VEL
LIN {X 0,Y 69.918,Z 464.434,A -85,B 0,C 180,E1 -27984.231,E2 -27984.231} C_VEL
LIN {X 0,Y 69.783,Z 464.586,A -85,B 0,C 180,E1 -27990,E2 -27990} C_VEL
LIN {X 0,Y 70.543,Z 464.027,A -85,B 0,C 180,E1 -28001.494,E2 -28001.494} C_VEL
LIN {X 0,Y 73.37,Z 462.357,A -85,B 0,C 180,E1 -28012.529,E2 -28012.529} C_VEL
LIN {X 0,Y 78.355,Z 459.53,A -85,B 0,C 180,E1 -28022.559,E2 -28022.559} C_VEL
LIN {X 0,Y 85.315,Z 455.474,A -85,B 0,C 180,E1 -28031.226,E2 -28031.226} C_VEL
LIN {X 0,Y 93.797,Z 450.089,A -85,B 0,C 180,E1 -28038.529,E2 -28038.529} C_VEL
LIN {X 0,Y 103.544,Z 443.217,A -85,B 0,C 180,E1 -28044.538,E2 -28044.538} C_VEL
LIN {X 0,Y 112.851,Z 435.828,A -85,B 0,C 180,E1 -28048.905,E2 -28048.905} C_VEL
LIN {X 0,Y 121.774,Z 427.626,A -85,B 0,C 180,E1 -28052.502,E2 -28052.502} C_VEL
LIN {X 0,Y 131.289,Z 417.828,A -85,B 0,C 180,E1 -28055.509,E2 -28055.509} C_VEL
LIN {X 0,Y 140.314,Z 407.096,A -85,B 0,C 180,E1 -28057.915,E2 -28057.915} C_VEL
LIN {X 0,Y 148.787,Z 395.373,A -85,B 0,C 180,E1 -28059.853,E2 -28059.853} C_VEL
LIN {X 0,Y 156.456,Z 382.775,A -85,B 0,C 180,E1 -28061.463,E2 -28061.463} C_VEL
LIN {X 0,Y 162.83,Z 370.187,A -85,B 0,C 180,E1 -28062.737,E2 -28062.737} C_VEL
LIN {X 0,Y 168.805,Z 355.749,A -85,B 0,C 180,E1 -28063.778,E2 -28063.778} C_VEL
LIN {X 0,Y 173.424,Z 341.434,A -85,B 0,C 180,E1 -28064.524,E2 -28064.524} C_VEL
LIN {X 0,Y 176.784,Z 327.285,A -85,B 0,C 180,E1 -28065.073,E2 -28065.073} C_VEL
LIN {X 0,Y 179.209,Z 311.307,A -85,B 0,C 180,E1 -28065.472,E2 -28065.472} C_VEL
LIN {X 0,Y 181.09,Z 293.388,A -85,B 0,C 180,E1 -28065.962,E2 -28065.962} C_VEL
LIN {X 0,Y 179.593,Z 289.326,A -85,B 0,C 180,E1 -28068.859,E2 -28068.859} C_VEL
LIN {X 0,Y 178.085,Z 285.006,A -85,B 0,C 180,E1 -28073.058,E2 -28073.058} C_VEL
LIN {X 0,Y 177.299,Z 281.498,A -85,B 0,C 180,E1 -28078.864,E2 -28078.864} C_VEL
LIN {X 0,Y 177.293,Z 281.726,A -85,B 0,C 180,E1 -28081.135,E2 -28081.135} C_VEL
LIN {X 0,Y 178.259,Z 285.553,A -85,B 0,C 180,E1 -28087.219,E2 -28087.219} C_VEL
LIN {X 0,Y 179.635,Z 289.345,A -85,B 0,C 180,E1 -28090.864,E2 -28090.864} C_VEL
LIN {X 0,Y 181.156,Z 293.558,A -85,B 0,C 180,E1 -28093.801,E2 -28093.801} C_VEL
LIN {X 0,Y 177.722,Z 322.993,A -85,B 0,C 180,E1 -28094.455,E2 -28094.455} C_VEL
LIN {X 0,Y 174.554,Z 338.53,A -85,B 0,C 180,E1 -28094.916,E2 -28094.916} C_VEL
LIN {X 0,Y 170.063,Z 353.733,A -85,B 0,C 180,E1 -28095.546,E2 -28095.546} C_VEL
LIN {X 0,Y 164.777,Z 367.446,A -85,B 0,C 180,E1 -28096.329,E2 -28096.329} C_VEL
LIN {X 0,Y 158.329,Z 380.884,A -85,B 0,C 180,E1 -28097.377,E2 -28097.377} C_VEL
LIN {X 0,Y 151.19,Z 393.282,A -85,B 0,C 180,E1 -28098.715,E2 -28098.715} C_VEL
LIN {X 0,Y 143.975,Z 403.987,A -85,B 0,C 180,E1 -28100.217,E2 -28100.217} C_VEL
LIN {X 0,Y 134.876,Z 415.589,A -85,B 0,C 180,E1 -28102.346,E2 -28102.346} C_VEL
LIN {X 0,Y 125.863,Z 425.548,A -85,B 0,C 180,E1 -28104.854,E2 -28104.854} C_VEL
LIN {X 0,Y 115.697,Z 435.297,A -85,B 0,C 180,E1 -28108.26,E2 -28108.26} C_VEL
LIN {X 0,Y 106.179,Z 443.445,A -85,B 0,C 180,E1 -28112.443,E2 -28112.443} C_VEL
LIN {X 0,Y 97.241,Z 450.189,A -85,B 0,C 180,E1 -28117.343,E2 -28117.343} C_VEL
LIN {X 0,Y 88.007,Z 456.417,A -85,B 0,C 180,E1 -28124.051,E2 -28124.051} C_VEL
LIN {X 0,Y 80.302,Z 461.246,A -85,B 0,C 180,E1 -28132.219,E2 -28132.219} C_VEL
LIN {X 0,Y 74.43,Z 464.793,A -85,B 0,C 180,E1 -28141.828,E2 -28141.828} C_VEL
LIN {X 0,Y 70.777,Z 467.137,A -85,B 0,C 180,E1 -28152.668,E2 -28152.668} C_VEL
LIN {X 0,Y 69.535,Z 468.328,A -85,B 0,C 180,E1 -28164.199,E2 -28164.199} C_VEL
LIN {X 0,Y 69.666,Z 468.491,A -85,B 0,C 180,E1 -28170,E2 -28170} C_VEL
LIN {X 0,Y 69.858,Z 467.853,A -85,B 0,C 180,E1 -28181.607,E2 -28181.607} C_VEL
LIN {X 0,Y 72.244,Z 466.058,A -85,B 0,C 180,E1 -28192.9,E2 -28192.9} C_VEL
LIN {X 0,Y 77.052,Z 463.096,A -85,B 0,C 180,E1 -28203.18,E2 -28203.18} C_VEL
LIN {X 0,Y 83.888,Z 458.897,A -85,B 0,C 180,E1 -28212.085,E2 -28212.085} C_VEL
LIN {X 0,Y 92.397,Z 453.352,A -85,B 0,C 180,E1 -28219.52,E2 -28219.52} C_VEL
LIN {X 0,Y 102.237,Z 446.315,A -85,B 0,C 180,E1 -28225.579,E2 -28225.579} C_VEL
LIN {X 0,Y 112.875,Z 437.563,A -85,B 0,C 180,E1 -28230.655,E2 -28230.655} C_VEL
LIN {X 0,Y 122.885,Z 428.279,A -85,B 0,C 180,E1 -28234.26,E2 -28234.26} C_VEL
LIN {X 0,Y 131.813,Z 418.85,A -85,B 0,C 180,E1 -28236.888,E2 -28236.888} C_VEL
LIN {X 0,Y 140.113,Z 408.837,A -85,B 0,C 180,E1 -28238.895,E2 -28238.895} C_VEL
LIN {X 0,Y 143.188,Z 404.464,A -85,B 0,C 180,E1 -28239.917,E2 -28239.917} C_VEL
LIN {X 0,Y 147.253,Z 397.213,A -85,B 0,C 180,E1 -28242.057,E2 -28242.057} C_VEL
LIN {X 0,Y 151.122,Z 389.649,A -85,B 0,C 180,E1 -28243.998,E2 -28243.998} C_VEL
LIN {X 0,Y 153.786,Z 384.725,A -85,B 0,C 180,E1 -28244.721,E2 -28244.721} C_VEL
LIN {X 0,Y 160.452,Z 371.946,A -85,B 0,C 180,E1 -28245.721,E2 -28245.721} C_VEL
LIN {X 0,Y 166.226,Z 358.399,A -85,B 0,C 180,E1 -28246.516,E2 -28246.516} C_VEL
LIN {X 0,Y 171.203,Z 343.379,A -85,B 0,C 180,E1 -28247.151,E2 -28247.151} C_VEL
LIN {X 0,Y 174.762,Z 328.465,A -85,B 0,C 180,E1 -28247.617,E2 -28247.617} C_VEL
LIN {X 0,Y 177.203,Z 312.114,A -85,B 0,C 180,E1 -28247.975,E2 -28247.975} C_VEL
LIN {X 0,Y 178.785,Z 297.712,A -85,B 0,C 180,E1 -28248.315,E2 -28248.315} C_VEL
LIN {X 0,Y 177.429,Z 293.76,A -85,B 0,C 180,E1 -28251.601,E2 -28251.601} C_VEL
LIN {X 0,Y 176.738,Z 291.599,A -85,B 0,C 180,E1 -28253.98,E2 -28253.98} C_VEL
LIN {X 0,Y 176.098,Z 288.421,A -85,B 0,C 180,E1 -28259.429,E2 -28259.429} C_VEL
LIN {X 0,Y 176.108,Z 288.691,A -85,B 0,C 180,E1 -28261.715,E2 -28261.715} C_VEL
LIN {X 0,Y 176.939,Z 292.338,A -85,B 0,C 180,E1 -28267.274,E2 -28267.274} C_VEL
LIN {X 0,Y 178.059,Z 295.716,A -85,B 0,C 180,E1 -28270.527,E2 -28270.527} C_VEL
LIN {X 0,Y 178.778,Z 297.783,A -85,B 0,C 180,E1 -28272.126,E2 -28272.126} C_VEL
LIN {X 0,Y 175.986,Z 320.823,A -85,B 0,C 180,E1 -28272.629,E2 -28272.629} C_VEL
LIN {X 0,Y 172.974,Z 335.535,A -85,B 0,C 180,E1 -28273.032,E2 -28273.032} C_VEL
LIN {X 0,Y 168.637,Z 350.455,A -85,B 0,C 180,E1 -28273.698,E2 -28273.698} C_VEL
LIN {X 0,Y 163.364,Z 364.237,A -85,B 0,C 180,E1 -28274.543,E2 -28274.543} C_VEL
LIN {X 0,Y 156.98,Z 377.619,A -85,B 0,C 180,E1 -28275.62,E2 -28275.62} C_VEL
LIN {X 0,Y 149.751,Z 390.208,A -85,B 0,C 180,E1 -28277.016,E2 -28277.016} C_VEL
LIN {X 0,Y 141.807,Z 401.766,A -85,B 0,C 180,E1 -28278.587,E2 -28278.587} C_VEL
LIN {X 0,Y 133.202,Z 412.503,A -85,B 0,C 180,E1 -28280.524,E2 -28280.524} C_VEL
LIN {X 0,Y 123.971,Z 422.431,A -85,B 0,C 180,E1 -28282.894,E2 -28282.894} C_VEL
LIN {X 0,Y 115.105,Z 430.857,A -85,B 0,C 180,E1 -28285.763,E2 -28285.763} C_VEL
LIN {X 0,Y 107.955,Z 436.886,A -85,B 0,C 180,E1 -28288.494,E2 -28288.494} C_VEL
LIN {X 0,Y 99.639,Z 443.186,A -85,B 0,C 180,E1 -28292.176,E2 -28292.176} C_VEL
LIN {X 0,Y 89.29,Z 450.11,A -85,B 0,C 180,E1 -28298.085,E2 -28298.085} C_VEL
LIN {X 0,Y 80.118,Z 455.539,A -85,B 0,C 180,E1 -28305.431,E2 -28305.431} C_VEL
LIN {X 0,Y 72.491,Z 459.627,A -85,B 0,C 180,E1 -28314.43,E2 -28314.43} C_VEL
LIN {X 0,Y 66.905,Z 462.487,A -85,B 0,C 180,E1 -28325.155,E2 -28325.155} C_VEL
LIN {X 0,Y 63.597,Z 464.196,A -85,B 0,C 180,E1 -28337.231,E2 -28337.231} C_VEL
LIN {X 0,Y 62.699,Z 464.784,A -85,B 0,C 180,E1 -28350,E2 -28350} C_VEL
LIN {X 0,Y 63.593,Z 464.225,A -85,B 0,C 180,E1 -28362.77,E2 -28362.77} C_VEL
LIN {X 0,Y 66.827,Z 462.557,A -85,B 0,C 180,E1 -28374.877,E2 -28374.877} C_VEL
LIN {X 0,Y 72.456,Z 459.729,A -85,B 0,C 180,E1 -28385.59,E2 -28385.59} C_VEL
LIN {X 0,Y 80.083,Z 455.673,A -85,B 0,C 180,E1 -28394.594,E2 -28394.594} C_VEL
LIN {X 0,Y 89.237,Z 450.287,A -85,B 0,C 180,E1 -28401.959,E2 -28401.959} C_VEL
LIN {X 0,Y 99.586,Z 443.414,A -85,B 0,C 180,E1 -28407.873,E2 -28407.873} C_VEL
LIN {X 0,Y 109.347,Z 436.025,A -85,B 0,C 180,E1 -28412.098,E2 -28412.098} C_VEL
LIN {X 0,Y 119.356,Z 427.19,A -85,B 0,C 180,E1 -28415.774,E2 -28415.774} C_VEL
LIN {X 0,Y 128.502,Z 418.025,A -85,B 0,C 180,E1 -28418.399,E2 -28418.399} C_VEL
LIN {X 0,Y 137.794,Z 407.292,A -85,B 0,C 180,E1 -28420.66,E2 -28420.66} C_VEL
LIN {X 0,Y 146.495,Z 395.568,A -85,B 0,C 180,E1 -28422.458,E2 -28422.458} C_VEL
LIN {X 0,Y 154.681,Z 382.365,A -85,B 0,C 180,E1 -28424.032,E2 -28424.032} C_VEL
LIN {X 0,Y 160.868,Z 370.38,A -85,B 0,C 180,E1 -28425.151,E2 -28425.151} C_VEL
LIN {X 0,Y 166.56,Z 357.067,A -85,B 0,C 180,E1 -28426.047,E2 -28426.047} C_VEL
LIN {X 0,Y 171.466,Z 342.383,A -85,B 0,C 180,E1 -28426.772,E2 -28426.772} C_VEL
LIN {X 0,Y 174.983,Z 327.995,A -85,B 0,C 180,E1 -28427.306,E2 -28427.306} C_VEL
LIN {X 0,Y 177.342,Z 313.23,A -85,B 0,C 180,E1 -28427.664,E2 -28427.664} C_VEL
LIN {X 0,Y 179.049,Z 297.995,A -85,B 0,C 180,E1 -28428,E2 -28428} C_VEL
LIN {X 0,Y 177.702,Z 294.067,A -85,B 0,C 180,E1 -28431.285,E2 -28431.285} C_VEL
LIN {X 0,Y 176.908,Z 291.591,A -85,B 0,C 180,E1 -28434.133,E2 -28434.133} C_VEL
LIN {X 0,Y 176.418,Z 288.511,A -85,B 0,C 180,E1 -28439.429,E2 -28439.429} C_VEL
LIN {X 0,Y 176.413,Z 288.749,A -85,B 0,C 180,E1 -28440.856,E2 -28440.856} C_VEL
LIN {X 0,Y 177.204,Z 292.414,A -85,B 0,C 180,E1 -28446.69,E2 -28446.69} C_VEL
LIN {X 0,Y 178.362,Z 295.93,A -85,B 0,C 180,E1 -28450.098,E2 -28450.098} C_VEL
LIN {X 0,Y 179.082,Z 298.017,A -85,B 0,C 180,E1 -28451.706,E2 -28451.706} C_VEL
LIN {X 0,Y 176.008,Z 323.222,A -85,B 0,C 180,E1 -28452.225,E2 -28452.225} C_VEL
LIN {X 0,Y 172.863,Z 338.341,A -85,B 0,C 180,E1 -28452.641,E2 -28452.641} C_VEL
LIN {X 0,Y 168.301,Z 353.542,A -85,B 0,C 180,E1 -28453.219,E2 -28453.219} C_VEL
LIN {X 0,Y 162.925,Z 367.254,A -85,B 0,C 180,E1 -28453.934,E2 -28453.934} C_VEL
LIN {X 0,Y 156.35,Z 380.689,A -85,B 0,C 180,E1 -28454.885,E2 -28454.885} C_VEL
LIN {X 0,Y 149.052,Z 393.086,A -85,B 0,C 180,E1 -28456.113,E2 -28456.113} C_VEL
LIN {X 0,Y 141.358,Z 404.2,A -85,B 0,C 180,E1 -28457.563,E2 -28457.563} C_VEL
LIN {X 0,Y 132.327,Z 415.392,A -85,B 0,C 180,E1 -28459.486,E2 -28459.486} C_VEL
LIN {X 0,Y 123.029,Z 425.35,A -85,B 0,C 180,E1 -28461.831,E2 -28461.831} C_VEL
LIN {X 0,Y 112.481,Z 435.098,A -85,B 0,C 180,E1 -28465.043,E2 -28465.043} C_VEL
LIN {X 0,Y 102.501,Z 443.245,A -85,B 0,C 180,E1 -28469.048,E2 -28469.048} C_VEL
LIN {X 0,Y 93.08,Z 449.99,A -85,B 0,C 180,E1 -28473.843,E2 -28473.843} C_VEL
LIN {X 0,Y 83.174,Z 456.217,A -85,B 0,C 180,E1 -28480.493,E2 -28480.493} C_VEL
LIN {X 0,Y 74.775,Z 461.047,A -85,B 0,C 180,E1 -28488.858,E2 -28488.858} C_VEL
LIN {X 0,Y 68.207,Z 464.593,A -85,B 0,C 180,E1 -28498.989,E2 -28498.989} C_VEL
LIN {X 0,Y 63.99,Z 466.937,A -85,B 0,C 180,E1 -28510.762,E2 -28510.762} C_VEL
LIN {X 0,Y 62.447,Z 468.128,A -85,B 0,C 180,E1 -28523.538,E2 -28523.538} C_VEL
LIN {X 0,Y 62.555,Z 468.291,A -85,B 0,C 180,E1 -28530,E2 -28530} C_VEL
LIN {X 0,Y 62.88,Z 467.652,A -85,B 0,C 180,E1 -28542.917,E2 -28542.917} C_VEL
LIN {X 0,Y 65.702,Z 465.857,A -85,B 0,C 180,E1 -28555.332,E2 -28555.332} C_VEL
LIN {X 0,Y 71.159,Z 462.895,A -85,B 0,C 180,E1 -28566.341,E2 -28566.341} C_VEL
LIN {X 0,Y 78.719,Z 458.695,A -85,B 0,C 180,E1 -28575.581,E2 -28575.581} C_VEL
LIN {X 0,Y 87.908,Z 453.15,A -85,B 0,C 180,E1 -28583.08,E2 -28583.08} C_VEL
LIN {X 0,Y 95.686,Z 448.006,A -85,B 0,C 180,E1 -28587.636,E2 -28587.636} C_VEL
LIN {X 0,Y 104.462,Z 441.46,A -85,B 0,C 180,E1 -28591.905,E2 -28591.905} C_VEL
LIN {X 0,Y 113.957,Z 433.613,A -85,B 0,C 180,E1 -28595.46,E2 -28595.46} C_VEL
LIN {X 0,Y 124.531,Z 423.559,A -85,B 0,C 180,E1 -28598.621,E2 -28598.621} C_VEL
LIN {X 0,Y 133.914,Z 413.294,A -85,B 0,C 180,E1 -28600.851,E2 -28600.851} C_VEL
LIN {X 0,Y 143.568,Z 400.86,A -85,B 0,C 180,E1 -28602.86,E2 -28602.86} C_VEL
LIN {X 0,Y 152.273,Z 387.397,A -85,B 0,C 180,E1 -28604.464,E2 -28604.464} C_VEL
LIN {X 0,Y 153.786,Z 384.725,A -85,B 0,C 180,E1 -28604.721,E2 -28604.721} C_VEL
LIN {X 0,Y 156.37,Z 379.752,A -85,B 0,C 180,E1 -28605.401,E2 -28605.401} C_VEL
LIN {X 0,Y 159.793,Z 371.541,A -85,B 0,C 180,E1 -28607.032,E2 -28607.032} C_VEL
LIN {X 0,Y 162.899,Z 363.103,A -85,B 0,C 180,E1 -28608.498,E2 -28608.498} C_VEL
LIN {X 0,Y 164.895,Z 357.711,A -85,B 0,C 180,E1 -28608.94,E2 -28608.94} C_VEL
LIN {X 0,Y 169.766,Z 343.171,A -85,B 0,C 180,E1 -28609.486,E2 -28609.486} C_VEL
LIN {X 0,Y 173.291,Z 328.741,A -85,B 0,C 180,E1 -28609.895,E2 -28609.895} C_VEL
LIN {X 0,Y 175.817,Z 312.269,A -85,B 0,C 180,E1 -28610.232,E2 -28610.232} C_VEL
LIN {X 0,Y 176.925,Z 302.47,A -85,B 0,C 180,E1 -28610.444,E2 -28610.444} C_VEL
LIN {X 0,Y 175.806,Z 298.686,A -85,B 0,C 180,E1 -28614.149,E2 -28614.149} C_VEL
LIN {X 0,Y 175.23,Z 295.493,A -85,B 0,C 180,E1 -28619.426,E2 -28619.426} C_VEL
LIN {X 0,Y 175.226,Z 295.705,A -85,B 0,C 180,E1 -28621.437,E2 -28621.437} C_VEL
LIN {X 0,Y 175.866,Z 299.04,A -85,B 0,C 180,E1 -28626.598,E2 -28626.598} C_VEL
LIN {X 0,Y 176.893,Z 302.479,A -85,B 0,C 180,E1 -28629.938,E2 -28629.938} C_VEL
LIN {X 0,Y 174.048,Z 323.867,A -85,B 0,C 180,E1 -28630.411,E2 -28630.411} C_VEL
LIN {X 0,Y 170.702,Z 338.727,A -85,B 0,C 180,E1 -28630.829,E2 -28630.829} C_VEL
LIN {X 0,Y 165.841,Z 354.107,A -85,B 0,C 180,E1 -28631.513,E2 -28631.513} C_VEL
LIN {X 0,Y 160.076,Z 368.056,A -85,B 0,C 180,E1 -28632.348,E2 -28632.348} C_VEL
LIN {X 0,Y 152.761,Z 382.253,A -85,B 0,C 180,E1 -28633.518,E2 -28633.518} C_VEL
LIN {X 0,Y 144.563,Z 395.273,A -85,B 0,C 180,E1 -28634.932,E2 -28634.932} C_VEL
LIN {X 0,Y 135.669,Z 407.074,A -85,B 0,C 180,E1 -28636.595,E2 -28636.595} C_VEL
LIN {X 0,Y 126.106,Z 417.872,A -85,B 0,C 180,E1 -28638.661,E2 -28638.661} C_VEL
LIN {X 0,Y 116.489,Z 427.23,A -85,B 0,C 180,E1 -28641.109,E2 -28641.109} C_VEL
LIN {X 0,Y 106.262,Z 435.971,A -85,B 0,C 180,E1 -28644.576,E2 -28644.576} C_VEL
LIN {X 0,Y 96.04,Z 443.387,A -85,B 0,C 180,E1 -28648.582,E2 -28648.582} C_VEL
LIN {X 0,Y 85.082,Z 450.31,A -85,B 0,C 180,E1 -28654.307,E2 -28654.307} C_VEL
LIN {X 0,Y 75.201,Z 455.74,A -85,B 0,C 180,E1 -28661.613,E2 -28661.613} C_VEL
LIN {X 0,Y 66.83,Z 459.827,A -85,B 0,C 180,E1 -28670.878,E2 -28670.878} C_VEL
LIN {X 0,Y 60.496,Z 462.688,A -85,B 0,C 180,E1 -28682.31,E2 -28682.31} C_VEL
LIN {X 0,Y 56.681,Z 464.396,A -85,B 0,C 180,E1 -28695.642,E2 -28695.642} C_VEL
LIN {X 0,Y 55.608,Z 464.983,A -85,B 0,C 180,E1 -28710,E2 -28710} C_VEL
LIN {X 0,Y 56.674,Z 464.424,A -85,B 0,C 180,E1 -28724.36,E2 -28724.36} C_VEL
LIN {X 0,Y 60.425,Z 462.756,A -85,B 0,C 180,E1 -28737.726,E2 -28737.726} C_VEL
LIN {X 0,Y 66.799,Z 459.928,A -85,B 0,C 180,E1 -28749.144,E2 -28749.144} C_VEL
LIN {X 0,Y 75.166,Z 455.871,A -85,B 0,C 180,E1 -28758.418,E2 -28758.418} C_VEL
LIN {X 0,Y 85.026,Z 450.485,A -85,B 0,C 180,E1 -28765.748,E2 -28765.748} C_VEL
LIN {X 0,Y 95.978,Z 443.613,A -85,B 0,C 180,E1 -28771.487,E2 -28771.487} C_VEL
LIN {X 0,Y 106.204,Z 436.223,A -85,B 0,C 180,E1 -28775.493,E2 -28775.493} C_VEL
LIN {X 0,Y 116.69,Z 427.32,A -85,B 0,C 180,E1 -28778.988,E2 -28778.988} C_VEL
LIN {X 0,Y 126.061,Z 418.221,A -85,B 0,C 180,E1 -28781.4,E2 -28781.4} C_VEL
LIN {X 0,Y 135.608,Z 407.488,A -85,B 0,C 180,E1 -28783.494,E2 -28783.494} C_VEL
LIN {X 0,Y 144.515,Z 395.763,A -85,B 0,C 180,E1 -28785.142,E2 -28785.142} C_VEL
LIN {X 0,Y 152.874,Z 382.56,A -85,B 0,C 180,E1 -28786.601,E2 -28786.601} C_VEL
LIN {X 0,Y 159.198,Z 370.572,A -85,B 0,C 180,E1 -28787.619,E2 -28787.619} C_VEL
LIN {X 0,Y 165.402,Z 356.132,A -85,B 0,C 180,E1 -28788.505,E2 -28788.505} C_VEL
LIN {X 0,Y 170.192,Z 341.811,A -85,B 0,C 180,E1 -28789.126,E2 -28789.126} C_VEL
LIN {X 0,Y 173.659,Z 327.723,A -85,B 0,C 180,E1 -28789.596,E2 -28789.596} C_VEL
LIN {X 0,Y 176.17,Z 311.81,A -85,B 0,C 180,E1 -28789.936,E2 -28789.936} C_VEL
LIN {X 0,Y 177.18,Z 302.711,A -85,B 0,C 180,E1 -28790.169,E2 -28790.169} C_VEL
LIN {X 0,Y 176.036,Z 298.726,A -85,B 0,C 180,E1 -28794.104,E2 -28794.104} C_VEL
LIN {X 0,Y 175.555,Z 295.539,A -85,B 0,C 180,E1 -28799.426,E2 -28799.426} C_VEL
LIN {X 0,Y 175.527,Z 296.033,A -85,B 0,C 180,E1 -28801.003,E2 -28801.003} C_VEL
LIN {X 0,Y 176.202,Z 299.374,A -85,B 0,C 180,E1 -28806.297,E2 -28806.297} C_VEL
LIN {X 0,Y 177.2,Z 302.738,A -85,B 0,C 180,E1 -28809.526,E2 -28809.526} C_VEL
LIN {X 0,Y 174.662,Z 322.95,A -85,B 0,C 180,E1 -28809.952,E2 -28809.952} C_VEL
LIN {X 0,Y 171.32,Z 338.616,A -85,B 0,C 180,E1 -28810.337,E2 -28810.337} C_VEL
LIN {X 0,Y 166.822,Z 353.35,A -85,B 0,C 180,E1 -28810.848,E2 -28810.848} C_VEL
LIN {X 0,Y 161.364,Z 367.061,A -85,B 0,C 180,E1 -28811.489,E2 -28811.489} C_VEL
LIN {X 0,Y 154.679,Z 380.495,A -85,B 0,C 180,E1 -28812.344,E2 -28812.344} C_VEL
LIN {X 0,Y 147.229,Z 392.89,A -85,B 0,C 180,E1 -28813.441,E2 -28813.441} C_VEL
LIN {X 0,Y 138.226,Z 405.513,A -85,B 0,C 180,E1 -28814.974,E2 -28814.974} C_VEL
LIN {X 0,Y 128.517,Z 416.985,A -85,B 0,C 180,E1 -28816.863,E2 -28816.863} C_VEL
LIN {X 0,Y 118.978,Z 426.644,A -85,B 0,C 180,E1 -28819.07,E2 -28819.07} C_VEL
LIN {X 0,Y 108.119,Z 436.139,A -85,B 0,C 180,E1 -28822.136,E2 -28822.136} C_VEL
LIN {X 0,Y 97.769,Z 444.062,A -85,B 0,C 180,E1 -28826.031,E2 -28826.031} C_VEL
LIN {X 0,Y 86.529,Z 451.463,A -85,B 0,C 180,E1 -28831.479,E2 -28831.479} C_VEL
LIN {X 0,Y 76.266,Z 457.341,A -85,B 0,C 180,E1 -28838.437,E2 -28838.437} C_VEL
LIN {X 0,Y 69.203,Z 461.007,A -85,B 0,C 180,E1 -28845.306,E2 -28845.306} C_VEL
LIN {X 0,Y 62.173,Z 464.393,A -85,B 0,C 180,E1 -28855.583,E2 -28855.583} C_VEL
LIN {X 0,Y 57.278,Z 466.737,A -85,B 0,C 180,E1 -28868.401,E2 -28868.401} C_VEL
LIN {X 0,Y 55.366,Z 467.928,A -85,B 0,C 180,E1 -28882.707,E2 -28882.707} C_VEL
LIN {X 0,Y 55.463,Z 468.093,A -85,B 0,C 180,E1 -28890,E2 -28890} C_VEL
LIN {X 0,Y 55.953,Z 467.453,A -85,B 0,C 180,E1 -28904.549,E2 -28904.549} C_VEL
LIN {X 0,Y 59.312,Z 465.656,A -85,B 0,C 180,E1 -28918.292,E2 -28918.292} C_VEL
LIN {X 0,Y 65.521,Z 462.693,A -85,B 0,C 180,E1 -28930.059,E2 -28930.059} C_VEL
LIN {X 0,Y 73.868,Z 458.493,A -85,B 0,C 180,E1 -28939.565,E2 -28939.565} C_VEL
LIN {X 0,Y 83.798,Z 452.948,A -85,B 0,C 180,E1 -28947.001,E2 -28947.001} C_VEL
LIN {X 0,Y 94.844,Z 445.908,A -85,B 0,C 180,E1 -28952.774,E2 -28952.774} C_VEL
LIN {X 0,Y 105.076,Z 438.385,A -85,B 0,C 180,E1 -28956.878,E2 -28956.878} C_VEL
LIN {X 0,Y 115.826,Z 429.329,A -85,B 0,C 180,E1 -28960.135,E2 -28960.135} C_VEL
LIN {X 0,Y 125.291,Z 420.087,A -85,B 0,C 180,E1 -28962.477,E2 -28962.477} C_VEL
LIN {X 0,Y 134.987,Z 409.207,A -85,B 0,C 180,E1 -28964.406,E2 -28964.406} C_VEL
LIN {X 0,Y 143.595,Z 397.812,A -85,B 0,C 180,E1 -28965.983,E2 -28965.983} C_VEL
LIN {X 0,Y 152.178,Z 384.332,A -85,B 0,C 180,E1 -28967.32,E2 -28967.32} C_VEL
LIN {X 0,Y 158.843,Z 371.741,A -85,B 0,C 180,E1 -28968.215,E2 -28968.215} C_VEL
LIN {X 0,Y 164.895,Z 357.711,A -85,B 0,C 180,E1 -28968.94,E2 -28968.94} C_VEL
LIN {X 0,Y 166.809,Z 352.231,A -85,B 0,C 180,E1 -28969.36,E2 -28969.36} C_VEL
LIN {X 0,Y 170.644,Z 336.177,A -85,B 0,C 180,E1 -28971.717,E2 -28971.717} C_VEL
LIN {X 0,Y 171.786,Z 330.543,A -85,B 0,C 180,E1 -28972.169,E2 -28972.169} C_VEL
LIN {X 0,Y 172.172,Z 328.618,A -85,B 0,C 180,E1 -28972.215,E2 -28972.215} C_VEL
LIN {X 0,Y 174.593,Z 313.405,A -85,B 0,C 180,E1 -28972.506,E2 -28972.506} C_VEL
LIN {X 0,Y 175.272,Z 307.418,A -85,B 0,C 180,E1 -28972.66,E2 -28972.66} C_VEL
LIN {X 0,Y 174.654,Z 305.105,A -85,B 0,C 180,E1 -28975.384,E2 -28975.384} C_VEL
LIN {X 0,Y 174.361,Z 302.569,A -85,B 0,C 180,E1 -28979.424,E2 -28979.424} C_VEL
LIN {X 0,Y 174.342,Z 302.781,A -85,B 0,C 180,E1 -28981.178,E2 -28981.178} C_VEL
LIN {X 0,Y 174.842,Z 305.899,A -85,B 0,C 180,E1 -28986.057,E2 -28986.057} C_VEL
LIN {X 0,Y 175.261,Z 307.434,A -85,B 0,C 180,E1 -28987.758,E2 -28987.758} C_VEL
LIN {X 0,Y 172.846,Z 324.408,A -85,B 0,C 180,E1 -28988.104,E2 -28988.104} C_VEL
LIN {X 0,Y 169.346,Z 339.554,A -85,B 0,C 180,E1 -28988.504,E2 -28988.504} C_VEL
LIN {X 0,Y 164.506,Z 354.496,A -85,B 0,C 180,E1 -28989.106,E2 -28989.106} C_VEL
LIN {X 0,Y 158.711,Z 368.26,A -85,B 0,C 180,E1 -28989.846,E2 -28989.846} C_VEL
LIN {X 0,Y 151.838,Z 381.467,A -85,B 0,C 180,E1 -28990.817,E2 -28990.817} C_VEL
LIN {X 0,Y 143.738,Z 394.305,A -85,B 0,C 180,E1 -28992.071,E2 -28992.071} C_VEL
LIN {X 0,Y 135.459,Z 405.333,A -85,B 0,C 180,E1 -28993.392,E2 -28993.392} C_VEL
LIN {X 0,Y 125.653,Z 416.444,A -85,B 0,C 180,E1 -28995.242,E2 -28995.242} C_VEL
LIN {X 0,Y 114.351,Z 427.233,A -85,B 0,C 180,E1 -28997.712,E2 -28997.712} C_VEL
LIN {X 0,Y 103.504,Z 436.172,A -85,B 0,C 180,E1 -29000.991,E2 -29000.991} C_VEL
LIN {X 0,Y 92.835,Z 443.589,A -85,B 0,C 180,E1 -29004.707,E2 -29004.707} C_VEL
LIN {X 0,Y 81.277,Z 450.511,A -85,B 0,C 180,E1 -29010.151,E2 -29010.151} C_VEL
LIN {X 0,Y 70.668,Z 455.941,A -85,B 0,C 180,E1 -29017.287,E2 -29017.287} C_VEL
LIN {X 0,Y 61.475,Z 460.027,A -85,B 0,C 180,E1 -29026.691,E2 -29026.691} C_VEL
LIN {X 0,Y 54.277,Z 462.888,A -85,B 0,C 180,E1 -29038.807,E2 -29038.807} C_VEL
LIN {X 0,Y 49.832,Z 464.595,A -85,B 0,C 180,E1 -29053.617,E2 -29053.617} C_VEL
LIN {X 0,Y 48.508,Z 465.182,A -85,B 0,C 180,E1 -29070,E2 -29070} C_VEL
LIN {X 0,Y 49.824,Z 464.623,A -85,B 0,C 180,E1 -29086.387,E2 -29086.387} C_VEL
LIN {X 0,Y 54.215,Z 462.955,A -85,B 0,C 180,E1 -29101.234,E2 -29101.234} C_VEL
LIN {X 0,Y 61.445,Z 460.126,A -85,B 0,C 180,E1 -29113.336,E2 -29113.336} C_VEL
LIN {X 0,Y 70.634,Z 456.07,A -85,B 0,C 180,E1 -29122.75,E2 -29122.75} C_VEL
LIN {X 0,Y 81.222,Z 450.684,A -85,B 0,C 180,E1 -29129.916,E2 -29129.916} C_VEL
LIN {X 0,Y 92.781,Z 443.811,A -85,B 0,C 180,E1 -29135.365,E2 -29135.365} C_VEL
LIN {X 0,Y 103.453,Z 436.42,A -85,B 0,C 180,E1 -29139.083,E2 -29139.083} C_VEL
LIN {X 0,Y 114.015,Z 427.784,A -85,B 0,C 180,E1 -29142.243,E2 -29142.243} C_VEL
LIN {X 0,Y 123.982,Z 418.417,A -85,B 0,C 180,E1 -29144.506,E2 -29144.506} C_VEL
LIN {X 0,Y 133.765,Z 407.684,A -85,B 0,C 180,E1 -29146.408,E2 -29146.408} C_VEL
LIN {X 0,Y 142.86,Z 395.958,A -85,B 0,C 180,E1 -29147.894,E2 -29147.894} C_VEL
LIN {X 0,Y 151.321,Z 382.859,A -85,B 0,C 180,E1 -29149.215,E2 -29149.215} C_VEL
LIN {X 0,Y 158.675,Z 369.003,A -85,B 0,C 180,E1 -29150.232,E2 -29150.232} C_VEL
LIN {X 0,Y 164.91,Z 354.261,A -85,B 0,C 180,E1 -29151.019,E2 -29151.019} C_VEL
LIN {X 0,Y 169.782,Z 339.148,A -85,B 0,C 180,E1 -29151.597,E2 -29151.597} C_VEL
LIN {X 0,Y 173.315,Z 323.615,A -85,B 0,C 180,E1 -29152.013,E2 -29152.013} C_VEL
LIN {X 0,Y 175.555,Z 307.725,A -85,B 0,C 180,E1 -29152.328,E2 -29152.328} C_VEL
LIN {X 0,Y 174.942,Z 305.332,A -85,B 0,C 180,E1 -29155.103,E2 -29155.103} C_VEL
LIN {X 0,Y 174.684,Z 302.599,A -85,B 0,C 180,E1 -29160,E2 -29160} C_VEL
LIN {X 0,Y 175.181,Z 306.187,A -85,B 0,C 180,E1 -29165.756,E2 -29165.756} C_VEL
LIN {X 0,Y 175.566,Z 307.673,A -85,B 0,C 180,E1 -29167.334,E2 -29167.334} C_VEL
LIN {X 0,Y 173.104,Z 325.318,A -85,B 0,C 180,E1 -29167.703,E2 -29167.703} C_VEL
LIN {X 0,Y 169.422,Z 341.18,A -85,B 0,C 180,E1 -29168.063,E2 -29168.063} C_VEL
LIN {X 0,Y 164.322,Z 356.638,A -85,B 0,C 180,E1 -29168.563,E2 -29168.563} C_VEL
LIN {X 0,Y 158.397,Z 370.422,A -85,B 0,C 180,E1 -29169.166,E2 -29169.166} C_VEL
LIN {X 0,Y 150.782,Z 384.647,A -85,B 0,C 180,E1 -29170.052,E2 -29170.052} C_VEL
LIN {X 0,Y 142.461,Z 397.451,A -85,B 0,C 180,E1 -29171.197,E2 -29171.197} C_VEL
LIN {X 0,Y 133.245,Z 409.353,A -85,B 0,C 180,E1 -29172.634,E2 -29172.634} C_VEL
LIN {X 0,Y 123.341,Z 420.179,A -85,B 0,C 180,E1 -29174.38,E2 -29174.38} C_VEL
LIN {X 0,Y 112.001,Z 430.73,A -85,B 0,C 180,E1 -29176.876,E2 -29176.876} C_VEL
LIN {X 0,Y 100.948,Z 439.518,A -85,B 0,C 180,E1 -29179.968,E2 -29179.968} C_VEL
LIN {X 0,Y 91.819,Z 445.894,A -85,B 0,C 180,E1 -29183.291,E2 -29183.291} C_VEL
LIN {X 0,Y 80.148,Z 452.888,A -85,B 0,C 180,E1 -29188.731,E2 -29188.731} C_VEL
LIN {X 0,Y 69.47,Z 458.398,A -85,B 0,C 180,E1 -29195.969,E2 -29195.969} C_VEL
LIN {X 0,Y 60.268,Z 462.574,A -85,B 0,C 180,E1 -29205.599,E2 -29205.599} C_VEL
LIN {X 0,Y 53.146,Z 465.51,A -85,B 0,C 180,E1 -29218.064,E2 -29218.064} C_VEL
LIN {X 0,Y 49.067,Z 467.275,A -85,B 0,C 180,E1 -29233.353,E2 -29233.353} C_VEL
LIN {X 0,Y 48.355,Z 467.894,A -85,B 0,C 180,E1 -29250,E2 -29250} C_VEL
LIN {X 0,Y 49.063,Z 467.252,A -85,B 0,C 180,E1 -29266.648,E2 -29266.648} C_VEL
LIN {X 0,Y 53.123,Z 465.456,A -85,B 0,C 180,E1 -29281.95,E2 -29281.95} C_VEL
LIN {X 0,Y 60.196,Z 462.491,A -85,B 0,C 180,E1 -29294.468,E2 -29294.468} C_VEL
LIN {X 0,Y 69.441,Z 458.292,A -85,B 0,C 180,E1 -29304.063,E2 -29304.063} C_VEL
LIN {X 0,Y 80.12,Z 452.746,A -85,B 0,C 180,E1 -29311.304,E2 -29311.304} C_VEL
LIN {X 0,Y 91.789,Z 445.706,A -85,B 0,C 180,E1 -29316.751,E2 -29316.751} C_VEL
LIN {X 0,Y 102.479,Z 438.183,A -85,B 0,C 180,E1 -29320.557,E2 -29320.557} C_VEL
LIN {X 0,Y 113.594,Z 429.126,A -85,B 0,C 180,E1 -29323.532,E2 -29323.532} C_VEL
LIN {X 0,Y 123.336,Z 419.885,A -85,B 0,C 180,E1 -29325.629,E2 -29325.629} C_VEL
LIN {X 0,Y 133.243,Z 409.004,A -85,B 0,C 180,E1 -29327.369,E2 -29327.369} C_VEL
LIN {X 0,Y 141.89,Z 397.812,A -85,B 0,C 180,E1 -29328.756,E2 -29328.756} C_VEL
LIN {X 0,Y 149.931,Z 385.558,A -85,B 0,C 180,E1 -29329.858,E2 -29329.858} C_VEL
LIN {X 0,Y 157.543,Z 371.536,A -85,B 0,C 180,E1 -29330.752,E2 -29330.752} C_VEL
LIN {X 0,Y 163.585,Z 357.756,A -85,B 0,C 180,E1 -29331.373,E2 -29331.373} C_VEL
LIN {X 0,Y 168.674,Z 342.748,A -85,B 0,C 180,E1 -29331.867,E2 -29331.867} C_VEL
LIN {X 0,Y 172.172,Z 328.618,A -85,B 0,C 180,E1 -29332.215,E2 -29332.215} C_VEL
LIN {X 0,Y 172.904,Z 324.442,A -85,B 0,C 180,E1 -29332.438,E2 -29332.438} C_VEL
LIN {X 0,Y 173.376,Z 320.49,A -85,B 0,C 180,E1 -29332.991,E2 -29332.991} C_VEL
LIN {X 0,Y 173.661,Z 315.898,A -85,B 0,C 180,E1 -29334.106,E2 -29334.106} C_VEL
LIN {X 0,Y 173.705,Z 313.247,A -85,B 0,C 180,E1 -29335.192,E2 -29335.192} C_VEL
LIN {X 0,Y 173.597,Z 311.68,A -85,B 0,C 180,E1 -29336.469,E2 -29336.469} C_VEL
LIN {X 0,Y 173.492,Z 309.515,A -85,B 0,C 180,E1 -29340,E2 -29340} C_VEL
LIN {X 0,Y 173.459,Z 310.731,A -85,B 0,C 180,E1 -29342.322,E2 -29342.322} C_VEL
LIN {X 0,Y 173.841,Z 312.747,A -85,B 0,C 180,E1 -29345.532,E2 -29345.532} C_VEL
LIN {X 0,Y 171.306,Z 328.234,A -85,B 0,C 180,E1 -29345.829,E2 -29345.829} C_VEL
LIN {X 0,Y 167.603,Z 342.761,A -85,B 0,C 180,E1 -29346.213,E2 -29346.213} C_VEL
LIN {X 0,Y 162.34,Z 357.847,A -85,B 0,C 180,E1 -29346.78,E2 -29346.78} C_VEL
LIN {X 0,Y 155.955,Z 371.985,A -85,B 0,C 180,E1 -29347.512,E2 -29347.512} C_VEL
LIN {X 0,Y 149.174,Z 384.181,A -85,B 0,C 180,E1 -29348.36,E2 -29348.36} C_VEL
LIN {X 0,Y 140.725,Z 396.847,A -85,B 0,C 180,E1 -29349.48,E2 -29349.48} C_VEL
LIN {X 0,Y 132.312,Z 407.478,A -85,B 0,C 180,E1 -29350.683,E2 -29350.683} C_VEL
LIN {X 0,Y 122.303,Z 418.275,A -85,B 0,C 180,E1 -29352.343,E2 -29352.343} C_VEL
LIN {X 0,Y 112.389,Z 427.435,A -85,B 0,C 180,E1 -29354.251,E2 -29354.251} C_VEL
LIN {X 0,Y 101.17,Z 436.373,A -85,B 0,C 180,E1 -29357.221,E2 -29357.221} C_VEL
LIN {X 0,Y 90.083,Z 443.79,A -85,B 0,C 180,E1 -29360.577,E2 -29360.577} C_VEL
LIN {X 0,Y 77.936,Z 450.712,A -85,B 0,C 180,E1 -29365.609,E2 -29365.609} C_VEL
LIN {X 0,Y 66.59,Z 456.141,A -85,B 0,C 180,E1 -29372.399,E2 -29372.399} C_VEL
LIN {X 0,Y 56.489,Z 460.228,A -85,B 0,C 180,E1 -29381.714,E2 -29381.714} C_VEL
LIN {X 0,Y 48.321,Z 463.088,A -85,B 0,C 180,E1 -29394.424,E2 -29394.424} C_VEL
LIN {X 0,Y 43.05,Z 464.794,A -85,B 0,C 180,E1 -29410.943,E2 -29410.943} C_VEL
LIN {X 0,Y 41.426,Z 465.38,A -85,B 0,C 180,E1 -29430,E2 -29430} C_VEL
LIN {X 0,Y 43.04,Z 464.822,A -85,B 0,C 180,E1 -29449.062,E2 -29449.062} C_VEL
LIN {X 0,Y 48.267,Z 463.154,A -85,B 0,C 180,E1 -29465.622,E2 -29465.622} C_VEL
LIN {X 0,Y 56.46,Z 460.325,A -85,B 0,C 180,E1 -29478.32,E2 -29478.32} C_VEL
LIN {X 0,Y 66.558,Z 456.269,A -85,B 0,C 180,E1 -29487.645,E2 -29487.645} C_VEL
LIN {X 0,Y 77.897,Z 450.882,A -85,B 0,C 180,E1 -29494.452,E2 -29494.452} C_VEL
LIN {X 0,Y 90.035,Z 444.01,A -85,B 0,C 180,E1 -29499.506,E2 -29499.506} C_VEL
LIN {X 0,Y 102.722,Z 435.422,A -85,B 0,C 180,E1 -29503.306,E2 -29503.306} C_VEL
LIN {X 0,Y 112.047,Z 427.981,A -85,B 0,C 180,E1 -29505.717,E2 -29505.717} C_VEL
LIN {X 0,Y 122.279,Z 418.613,A -85,B 0,C 180,E1 -29507.71,E2 -29507.71} C_VEL
LIN {X 0,Y 132.277,Z 407.879,A -85,B 0,C 180,E1 -29509.398,E2 -29509.398} C_VEL
LIN {X 0,Y 141.541,Z 396.153,A -85,B 0,C 180,E1 -29510.705,E2 -29510.705} C_VEL
LIN {X 0,Y 149.928,Z 383.434,A -85,B 0,C 180,E1 -29511.848,E2 -29511.848} C_VEL
LIN {X 0,Y 156.771,Z 370.958,A -85,B 0,C 180,E1 -29512.686,E2 -29512.686} C_VEL
LIN {X 0,Y 162.743,Z 357.642,A -85,B 0,C 180,E1 -29513.34,E2 -29513.34} C_VEL
LIN {X 0,Y 167.958,Z 342.674,A -85,B 0,C 180,E1 -29513.862,E2 -29513.862} C_VEL
LIN {X 0,Y 171.616,Z 328.352,A -85,B 0,C 180,E1 -29514.241,E2 -29514.241} C_VEL
LIN {X 0,Y 174.134,Z 313.027,A -85,B 0,C 180,E1 -29514.572,E2 -29514.572} C_VEL
LIN {X 0,Y 173.782,Z 309.98,A -85,B 0,C 180,E1 -29519.42,E2 -29519.42} C_VEL
LIN {X 0,Y 173.784,Z 309.975,A -85,B 0,C 180,E1 -29520.289,E2 -29520.289} C_VEL
LIN {X 0,Y 174.162,Z 312.959,A -85,B 0,C 180,E1 -29525.147,E2 -29525.147} C_VEL
LIN {X 0,Y 171.508,Z 329.303,A -85,B 0,C 180,E1 -29525.446,E2 -29525.446} C_VEL
LIN {X 0,Y 167.49,Z 344.786,A -85,B 0,C 180,E1 -29525.769,E2 -29525.769} C_VEL
LIN {X 0,Y 162.158,Z 359.716,A -85,B 0,C 180,E1 -29526.213,E2 -29526.213} C_VEL
LIN {X 0,Y 155.703,Z 373.755,A -85,B 0,C 180,E1 -29526.773,E2 -29526.773} C_VEL
LIN {X 0,Y 147.991,Z 387.303,A -85,B 0,C 180,E1 -29527.543,E2 -29527.543} C_VEL
LIN {X 0,Y 139.412,Z 399.799,A -85,B 0,C 180,E1 -29528.582,E2 -29528.582} C_VEL
LIN {X 0,Y 130.187,Z 411.116,A -85,B 0,C 180,E1 -29529.864,E2 -29529.864} C_VEL
LIN {X 0,Y 120.087,Z 421.615,A -85,B 0,C 180,E1 -29531.395,E2 -29531.395} C_VEL
LIN {X 0,Y 108.491,Z 431.893,A -85,B 0,C 180,E1 -29533.664,E2 -29533.664} C_VEL
LIN {X 0,Y 97.12,Z 440.443,A -85,B 0,C 180,E1 -29536.497,E2 -29536.497} C_VEL
LIN {X 0,Y 86.121,Z 447.568,A -85,B 0,C 180,E1 -29540.203,E2 -29540.203} C_VEL
LIN {X 0,Y 74.003,Z 454.18,A -85,B 0,C 180,E1 -29545.549,E2 -29545.549} C_VEL
LIN {X 0,Y 62.844,Z 459.365,A -85,B 0,C 180,E1 -29552.991,E2 -29552.991} C_VEL
LIN {X 0,Y 55.369,Z 462.374,A -85,B 0,C 180,E1 -29560.396,E2 -29560.396} C_VEL
LIN {X 0,Y 47.232,Z 465.31,A -85,B 0,C 180,E1 -29573.473,E2 -29573.473} C_VEL
LIN {X 0,Y 42.273,Z 467.075,A -85,B 0,C 180,E1 -29590.579,E2 -29590.579} C_VEL
LIN {X 0,Y 41.264,Z 467.695,A -85,B 0,C 180,E1 -29610,E2 -29610} C_VEL
LIN {X 0,Y 42.269,Z 467.052,A -85,B 0,C 180,E1 -29629.423,E2 -29629.423} C_VEL
LIN {X 0,Y 47.209,Z 465.255,A -85,B 0,C 180,E1 -29646.547,E2 -29646.547} C_VEL
LIN {X 0,Y 55.301,Z 462.29,A -85,B 0,C 180,E1 -29659.686,E2 -29659.686} C_VEL
LIN {X 0,Y 65.491,Z 458.09,A -85,B 0,C 180,E1 -29669.148,E2 -29669.148} C_VEL
LIN {X 0,Y 76.937,Z 452.544,A -85,B 0,C 180,E1 -29675.991,E2 -29675.991} C_VEL
LIN {X 0,Y 89.203,Z 445.504,A -85,B 0,C 180,E1 -29680.987,E2 -29680.987} C_VEL
LIN {X 0,Y 100.326,Z 437.981,A -85,B 0,C 180,E1 -29684.41,E2 -29684.41} C_VEL
LIN {X 0,Y 111.776,Z 428.924,A -85,B 0,C 180,E1 -29687.053,E2 -29687.053} C_VEL
LIN {X 0,Y 121.76,Z 419.683,A -85,B 0,C 180,E1 -29688.885,E2 -29688.885} C_VEL
LIN {X 0,Y 131.863,Z 408.801,A -85,B 0,C 180,E1 -29690.405,E2 -29690.405} C_VEL
LIN {X 0,Y 141.266,Z 396.793,A -85,B 0,C 180,E1 -29691.672,E2 -29691.672} C_VEL
LIN {X 0,Y 149.7,Z 383.925,A -85,B 0,C 180,E1 -29692.64,E2 -29692.64} C_VEL
LIN {X 0,Y 157.419,Z 369.563,A -85,B 0,C 180,E1 -29693.392,E2 -29693.392} C_VEL
LIN {X 0,Y 163.296,Z 355.915,A -85,B 0,C 180,E1 -29693.897,E2 -29693.897} C_VEL
LIN {X 0,Y 168.466,Z 340.246,A -85,B 0,C 180,E1 -29694.315,E2 -29694.315} C_VEL
LIN {X 0,Y 171.924,Z 325.395,A -85,B 0,C 180,E1 -29694.61,E2 -29694.61} C_VEL
LIN {X 0,Y 173.851,Z 312.681,A -85,B 0,C 180,E1 -29694.901,E2 -29694.901} C_VEL
LIN {X 0,Y 173.597,Z 311.68,A -85,B 0,C 180,E1 -29696.469,E2 -29696.469} C_VEL
LIN {X 0,Y 173.391,Z 311.673,A -85,B 0,C 180,E1 -29697.754,E2 -29697.754} C_VEL
LIN {X 0,Y 173.135,Z 312.768,A -85,B 0,C 180,E1 -29699.011,E2 -29699.011} C_VEL
LIN {X 0,Y 172.512,Z 317.969,A -85,B 0,C 180,E1 -29702.721,E2 -29702.721} C_VEL
LIN {X 0,Y 172.517,Z 318.352,A -85,B 0,C 180,E1 -29703.161,E2 -29703.161} C_VEL
LIN {X 0,Y 172.521,Z 318.415,A -85,B 0,C 180,E1 -29703.245,E2 -29703.245} C_VEL
LIN {X 0,Y 170.896,Z 327.6,A -85,B 0,C 180,E1 -29703.445,E2 -29703.445} C_VEL
LIN {X 0,Y 167.047,Z 342.749,A -85,B 0,C 180,E1 -29703.792,E2 -29703.792} C_VEL
LIN {X 0,Y 161.657,Z 358.052,A -85,B 0,C 180,E1 -29704.284,E2 -29704.284} C_VEL
LIN {X 0,Y 155.186,Z 372.19,A -85,B 0,C 180,E1 -29704.908,E2 -29704.908} C_VEL
LIN {X 0,Y 147.45,Z 385.806,A -85,B 0,C 180,E1 -29705.745,E2 -29705.745} C_VEL
LIN {X 0,Y 138.876,Z 398.219,A -85,B 0,C 180,E1 -29706.71,E2 -29706.71} C_VEL
LIN {X 0,Y 129.481,Z 409.622,A -85,B 0,C 180,E1 -29707.871,E2 -29707.871} C_VEL
LIN {X 0,Y 119.287,Z 420.097,A -85,B 0,C 180,E1 -29709.299,E2 -29709.299} C_VEL
LIN {X 0,Y 107.508,Z 430.324,A -85,B 0,C 180,E1 -29711.31,E2 -29711.31} C_VEL
LIN {X 0,Y 95.994,Z 438.798,A -85,B 0,C 180,E1 -29714.053,E2 -29714.053} C_VEL
LIN {X 0,Y 84.616,Z 445.855,A -85,B 0,C 180,E1 -29717.222,E2 -29717.222} C_VEL
LIN {X 0,Y 72.027,Z 452.395,A -85,B 0,C 180,E1 -29722.035,E2 -29722.035} C_VEL
LIN {X 0,Y 60.169,Z 457.495,A -85,B 0,C 180,E1 -29728.833,E2 -29728.833} C_VEL
LIN {X 0,Y 52.011,Z 460.429,A -85,B 0,C 180,E1 -29735.83,E2 -29735.83} C_VEL
LIN {X 0,Y 42.73,Z 463.288,A -85,B 0,C 180,E1 -29748.86,E2 -29748.86} C_VEL
LIN {X 0,Y 36.408,Z 464.993,A -85,B 0,C 180,E1 -29767.29,E2 -29767.29} C_VEL
LIN {X 0,Y 34.328,Z 465.579,A -85,B 0,C 180,E1 -29790.001,E2 -29790.001} C_VEL
LIN {X 0,Y 36.397,Z 465.021,A -85,B 0,C 180,E1 -29812.718,E2 -29812.718} C_VEL
LIN {X 0,Y 42.668,Z 463.353,A -85,B 0,C 180,E1 -29831.213,E2 -29831.213} C_VEL
LIN {X 0,Y 51.985,Z 460.525,A -85,B 0,C 180,E1 -29844.21,E2 -29844.21} C_VEL
LIN {X 0,Y 63.018,Z 456.468,A -85,B 0,C 180,E1 -29853.152,E2 -29853.152} C_VEL
LIN {X 0,Y 75.094,Z 451.081,A -85,B 0,C 180,E1 -29859.375,E2 -29859.375} C_VEL
LIN {X 0,Y 87.789,Z 444.208,A -85,B 0,C 180,E1 -29863.878,E2 -29863.878} C_VEL
LIN {X 0,Y 100.906,Z 435.62,A -85,B 0,C 180,E1 -29867.185,E2 -29867.185} C_VEL
LIN {X 0,Y 110.839,Z 427.909,A -85,B 0,C 180,E1 -29869.363,E2 -29869.363} C_VEL
LIN {X 0,Y 120.968,Z 418.809,A -85,B 0,C 180,E1 -29870.996,E2 -29870.996} C_VEL
LIN {X 0,Y 131.157,Z 408.075,A -85,B 0,C 180,E1 -29872.447,E2 -29872.447} C_VEL
LIN {X 0,Y 140.569,Z 396.348,A -85,B 0,C 180,E1 -29873.563,E2 -29873.563} C_VEL
LIN {X 0,Y 149.514,Z 382.919,A -85,B 0,C 180,E1 -29874.605,E2 -29874.605} C_VEL
LIN {X 0,Y 156.893,Z 369.389,A -85,B 0,C 180,E1 -29875.34,E2 -29875.34} C_VEL
LIN {X 0,Y 162.732,Z 356.116,A -85,B 0,C 180,E1 -29875.89,E2 -29875.89} C_VEL
LIN {X 0,Y 167.758,Z 341.417,A -85,B 0,C 180,E1 -29876.324,E2 -29876.324} C_VEL
LIN {X 0,Y 171.475,Z 326.332,A -85,B 0,C 180,E1 -29876.643,E2 -29876.643} C_VEL
LIN {X 0,Y 172.825,Z 318.664,A -85,B 0,C 180,E1 -29876.814,E2 -29876.814} C_VEL
LIN {X 0,Y 172.839,Z 316.983,A -85,B 0,C 180,E1 -29880,E2 -29880} C_VEL
LIN {X 0,Y 172.84,Z 318.687,A -85,B 0,C 180,E1 -29882.877,E2 -29882.877} C_VEL
LIN {X 0,Y 169.938,Z 333.526,A -85,B 0,C 180,E1 -29883.135,E2 -29883.135} C_VEL
LIN {X 0,Y 165.666,Z 348.376,A -85,B 0,C 180,E1 -29883.427,E2 -29883.427} C_VEL
LIN {X 0,Y 160.241,Z 362.515,A -85,B 0,C 180,E1 -29883.802,E2 -29883.802} C_VEL
LIN {X 0,Y 153.289,Z 376.744,A -85,B 0,C 180,E1 -29884.286,E2 -29884.286} C_VEL
LIN {X 0,Y 145.496,Z 389.715,A -85,B 0,C 180,E1 -29884.948,E2 -29884.948} C_VEL
LIN {X 0,Y 136.768,Z 401.842,A -85,B 0,C 180,E1 -29885.846,E2 -29885.846} C_VEL
LIN {X 0,Y 127.437,Z 412.816,A -85,B 0,C 180,E1 -29886.934,E2 -29886.934} C_VEL
LIN {X 0,Y 117.183,Z 423.049,A -85,B 0,C 180,E1 -29888.274,E2 -29888.274} C_VEL
LIN {X 0,Y 105.343,Z 433.052,A -85,B 0,C 180,E1 -29890.243,E2 -29890.243} C_VEL
LIN {X 0,Y 93.681,Z 441.368,A -85,B 0,C 180,E1 -29892.767,E2 -29892.767} C_VEL
LIN {X 0,Y 80.703,Z 449.193,A -85,B 0,C 180,E1 -29896.676,E2 -29896.676} C_VEL
LIN {X 0,Y 68.129,Z 455.418,A -85,B 0,C 180,E1 -29901.809,E2 -29901.809} C_VEL
LIN {X 0,Y 56.399,Z 460.245,A -85,B 0,C 180,E1 -29909.274,E2 -29909.274} C_VEL
LIN {X 0,Y 46.046,Z 463.792,A -85,B 0,C 180,E1 -29920.257,E2 -29920.257} C_VEL
LIN {X 0,Y 38.115,Z 466.135,A -85,B 0,C 180,E1 -29936.414,E2 -29936.414} C_VEL
LIN {X 0,Y 34.255,Z 467.33,A -85,B 0,C 180,E1 -29958.16,E2 -29958.16} C_VEL
LIN {X 0,Y 34.142,Z 467.496,A -85,B 0,C 180,E1 -29969.999,E2 -29969.999} C_VEL
LIN {X 0,Y 35.603,Z 466.851,A -85,B 0,C 180,E1 -29993.253,E2 -29993.253} C_VEL
LIN {X 0,Y 41.663,Z 465.054,A -85,B 0,C 180,E1 -30012.435,E2 -30012.435} C_VEL
LIN {X 0,Y 50.945,Z 462.088,A -85,B 0,C 180,E1 -30025.865,E2 -30025.865} C_VEL
LIN {X 0,Y 62.116,Z 457.888,A -85,B 0,C 180,E1 -30034.843,E2 -30034.843} C_VEL
LIN {X 0,Y 74.311,Z 452.342,A -85,B 0,C 180,E1 -30041.041,E2 -30041.041} C_VEL
LIN {X 0,Y 87.134,Z 445.302,A -85,B 0,C 180,E1 -30045.442,E2 -30045.442} C_VEL
LIN {X 0,Y 98.64,Z 437.779,A -85,B 0,C 180,E1 -30048.428,E2 -30048.428} C_VEL
LIN {X 0,Y 110.395,Z 428.722,A -85,B 0,C 180,E1 -30050.667,E2 -30050.667} C_VEL
LIN {X 0,Y 120.589,Z 419.48,A -85,B 0,C 180,E1 -30052.211,E2 -30052.211} C_VEL
LIN {X 0,Y 130.861,Z 408.597,A -85,B 0,C 180,E1 -30053.496,E2 -30053.496} C_VEL
LIN {X 0,Y 140.325,Z 396.706,A -85,B 0,C 180,E1 -30054.546,E2 -30054.546} C_VEL
LIN {X 0,Y 148.958,Z 383.722,A -85,B 0,C 180,E1 -30055.347,E2 -30055.347} C_VEL
LIN {X 0,Y 156.76,Z 369.358,A -85,B 0,C 180,E1 -30055.976,E2 -30055.976} C_VEL
LIN {X 0,Y 162.609,Z 355.931,A -85,B 0,C 180,E1 -30056.379,E2 -30056.379} C_VEL
LIN {X 0,Y 167.836,Z 340.297,A -85,B 0,C 180,E1 -30056.726,E2 -30056.726} C_VEL
LIN {X 0,Y 171.39,Z 325.251,A -85,B 0,C 180,E1 -30056.975,E2 -30056.975} C_VEL
LIN {X 0,Y 172.54,Z 318.455,A -85,B 0,C 180,E1 -30057.115,E2 -30057.115} C_VEL
LIN {X 0,Y 172.549,Z 316.623,A -85,B 0,C 180,E1 -30060,E2 -30060} C_VEL
LIN {X 0,Y 172.517,Z 318.352,A -85,B 0,C 180,E1 -30063.161,E2 -30063.161} C_VEL
LIN {X 0,Y 172.452,Z 319.411,A -85,B 0,C 180,E1 -30063.653,E2 -30063.653} C_VEL
LIN {X 0,Y 172.092,Z 321.904,A -85,B 0,C 180,E1 -30063.997,E2 -30063.997} C_VEL
LIN {X 0,Y 171.432,Z 325.341,A -85,B 0,C 180,E1 -30063.966,E2 -30063.966} C_VEL
LIN {X 0,Y 170.201,Z 330.669,A -85,B 0,C 180,E1 -30063.413,E2 -30063.413} C_VEL
LIN {X 0,Y 167.133,Z 341.688,A -85,B 0,C 180,E1 -30061.803,E2 -30061.803} C_VEL
LIN {X 0,Y 165.691,Z 346.232,A -85,B 0,C 180,E1 -30061.49,E2 -30061.49} C_VEL
LIN {X 0,Y 164.905,Z 348.529,A -85,B 0,C 180,E1 -30061.5,E2 -30061.5} C_VEL
LIN {X 0,Y 159.974,Z 361.3,A -85,B 0,C 180,E1 -30061.882,E2 -30061.882} C_VEL
LIN {X 0,Y 153.095,Z 375.449,A -85,B 0,C 180,E1 -30062.433,E2 -30062.433} C_VEL
LIN {X 0,Y 145.173,Z 388.649,A -85,B 0,C 180,E1 -30063.154,E2 -30063.154} C_VEL
LIN {X 0,Y 136.491,Z 400.649,A -85,B 0,C 180,E1 -30063.946,E2 -30063.946} C_VEL
LIN {X 0,Y 126.971,Z 411.738,A -85,B 0,C 180,E1 -30064.917,E2 -30064.917} C_VEL
LIN {X 0,Y 116.625,Z 421.919,A -85,B 0,C 180,E1 -30066.11,E2 -30066.11} C_VEL
LIN {X 0,Y 105.725,Z 431.011,A -85,B 0,C 180,E1 -30067.64,E2 -30067.64} C_VEL
LIN {X 0,Y 94.522,Z 438.998,A -85,B 0,C 180,E1 -30069.875,E2 -30069.875} C_VEL
LIN {X 0,Y 82.783,Z 446.056,A -85,B 0,C 180,E1 -30072.495,E2 -30072.495} C_VEL
LIN {X 0,Y 69.671,Z 452.595,A -85,B 0,C 180,E1 -30076.603,E2 -30076.603} C_VEL
LIN {X 0,Y 57.072,Z 457.696,A -85,B 0,C 180,E1 -30082.547,E2 -30082.547} C_VEL
LIN {X 0,Y 48.181,Z 460.629,A -85,B 0,C 180,E1 -30088.931,E2 -30088.931} C_VEL
LIN {X 0,Y 37.649,Z 463.488,A -85,B 0,C 180,E1 -30101.696,E2 -30101.696} C_VEL
LIN {X 0,Y 29.965,Z 465.193,A -85,B 0,C 180,E1 -30122.026,E2 -30122.026} C_VEL
LIN {X 0,Y 27.245,Z 465.777,A -85,B 0,C 180,E1 -30150.001,E2 -30150.001} C_VEL
LIN {X 0,Y 29.954,Z 465.22,A -85,B 0,C 180,E1 -30177.986,E2 -30177.986} C_VEL
LIN {X 0,Y 37.6,Z 463.553,A -85,B 0,C 180,E1 -30198.389,E2 -30198.389} C_VEL
LIN {X 0,Y 48.16,Z 460.724,A -85,B 0,C 180,E1 -30211.116,E2 -30211.116} C_VEL
LIN {X 0,Y 61.363,Z 456.179,A -85,B 0,C 180,E1 -30219.903,E2 -30219.903} C_VEL
LIN {X 0,Y 72.883,Z 451.28,A -85,B 0,C 180,E1 -30224.642,E2 -30224.642} C_VEL
LIN {X 0,Y 86.079,Z 444.407,A -85,B 0,C 180,E1 -30228.453,E2 -30228.453} C_VEL
LIN {X 0,Y 97.875,Z 437.014,A -85,B 0,C 180,E1 -30230.871,E2 -30230.871} C_VEL
LIN {X 0,Y 109.748,Z 428.107,A -85,B 0,C 180,E1 -30233.023,E2 -30233.023} C_VEL
LIN {X 0,Y 120.059,Z 419.006,A -85,B 0,C 180,E1 -30234.357,E2 -30234.357} C_VEL
LIN {X 0,Y 130.414,Z 408.27,A -85,B 0,C 180,E1 -30235.541,E2 -30235.541} C_VEL
LIN {X 0,Y 139.95,Z 396.543,A -85,B 0,C 180,E1 -30236.454,E2 -30236.454} C_VEL
LIN {X 0,Y 148.627,Z 383.745,A -85,B 0,C 180,E1 -30237.289,E2 -30237.289} C_VEL
LIN {X 0,Y 155.603,Z 371.344,A -85,B 0,C 180,E1 -30237.87,E2 -30237.87} C_VEL
LIN {X 0,Y 161.713,Z 358.024,A -85,B 0,C 180,E1 -30238.335,E2 -30238.335} C_VEL
LIN {X 0,Y 167.09,Z 342.871,A -85,B 0,C 180,E1 -30238.717,E2 -30238.717} C_VEL
LIN {X 0,Y 170.779,Z 328.713,A -85,B 0,C 180,E1 -30238.973,E2 -30238.973} C_VEL
LIN {X 0,Y 171.594,Z 324.489,A -85,B 0,C 180,E1 -30239.091,E2 -30239.091} C_VEL
LIN {X 0,Y 171.654,Z 324.137,A -85,B 0,C 180,E1 -30240,E2 -30240} C_VEL
LIN {X 0,Y 171.602,Z 324.501,A -85,B 0,C 180,E1 -30240.605,E2 -30240.605} C_VEL
LIN {X 0,Y 168.098,Z 339.452,A -85,B 0,C 180,E1 -30240.822,E2 -30240.822} C_VEL
LIN {X 0,Y 163.426,Z 353.726,A -85,B 0,C 180,E1 -30241.064,E2 -30241.064} C_VEL
LIN {X 0,Y 157.299,Z 368.074,A -85,B 0,C 180,E1 -30241.393,E2 -30241.393} C_VEL
LIN {X 0,Y 150.299,Z 381.207,A -85,B 0,C 180,E1 -30241.805,E2 -30241.805} C_VEL
LIN {X 0,Y 141.566,Z 394.599,A -85,B 0,C 180,E1 -30242.424,E2 -30242.424} C_VEL
LIN {X 0,Y 131.93,Z 406.867,A -85,B 0,C 180,E1 -30243.239,E2 -30243.239} C_VEL
LIN {X 0,Y 121.567,Z 417.954,A -85,B 0,C 180,E1 -30244.24,E2 -30244.24} C_VEL
LIN {X 0,Y 111.192,Z 427.345,A -85,B 0,C 180,E1 -30245.439,E2 -30245.439} C_VEL
LIN {X 0,Y 99.165,Z 436.583,A -85,B 0,C 180,E1 -30247.157,E2 -30247.157} C_VEL
LIN {X 0,Y 87.762,Z 443.993,A -85,B 0,C 180,E1 -30249.39,E2 -30249.39} C_VEL
LIN {X 0,Y 75.628,Z 450.666,A -85,B 0,C 180,E1 -30252.642,E2 -30252.642} C_VEL
LIN {X 0,Y 62.595,Z 456.541,A -85,B 0,C 180,E1 -30257.377,E2 -30257.377} C_VEL
LIN {X 0,Y 49.741,Z 461.227,A -85,B 0,C 180,E1 -30265.079,E2 -30265.079} C_VEL
LIN {X 0,Y 41.771,Z 463.592,A -85,B 0,C 180,E1 -30272.726,E2 -30272.726} C_VEL
LIN {X 0,Y 32.388,Z 465.935,A -85,B 0,C 180,E1 -30289.384,E2 -30289.384} C_VEL
LIN {X 0,Y 27.318,Z 467.13,A -85,B 0,C 180,E1 -30315.092,E2 -30315.092} C_VEL
LIN {X 0,Y 27.028,Z 467.297,A -85,B 0,C 180,E1 -30329.999,E2 -30329.999} C_VEL
LIN {X 0,Y 29.156,Z 466.651,A -85,B 0,C 180,E1 -30358.822,E2 -30358.822} C_VEL
LIN {X 0,Y 36.691,Z 464.852,A -85,B 0,C 180,E1 -30380.012,E2 -30380.012} C_VEL
LIN {X 0,Y 48.952,Z 461.366,A -85,B 0,C 180,E1 -30394.488,E2 -30394.488} C_VEL
LIN {X 0,Y 62.579,Z 456.429,A -85,B 0,C 180,E1 -30402.669,E2 -30402.669} C_VEL
LIN {X 0,Y 75.614,Z 450.513,A -85,B 0,C 180,E1 -30407.405,E2 -30407.405} C_VEL
LIN {X 0,Y 89.971,Z 442.464,A -85,B 0,C 180,E1 -30411.116,E2 -30411.116} C_VEL
LIN {X 0,Y 102.59,Z 433.873,A -85,B 0,C 180,E1 -30413.381,E2 -30413.381} C_VEL
LIN {X 0,Y 114.637,Z 424.079,A -85,B 0,C 180,E1 -30415.026,E2 -30415.026} C_VEL
LIN {X 0,Y 125.038,Z 414.071,A -85,B 0,C 180,E1 -30416.091,E2 -30416.091} C_VEL
LIN {X 0,Y 135.29,Z 402.398,A -85,B 0,C 180,E1 -30417.061,E2 -30417.061} C_VEL
LIN {X 0,Y 144.181,Z 390.327,A -85,B 0,C 180,E1 -30417.798,E2 -30417.798} C_VEL
LIN {X 0,Y 152.048,Z 377.523,A -85,B 0,C 180,E1 -30418.302,E2 -30418.302} C_VEL
LIN {X 0,Y 159.049,Z 363.541,A -85,B 0,C 180,E1 -30418.708,E2 -30418.708} C_VEL
LIN {X 0,Y 164.551,Z 349.695,A -85,B 0,C 180,E1 -30418.991,E2 -30418.991} C_VEL
LIN {X 0,Y 168.928,Z 335.155,A -85,B 0,C 180,E1 -30419.216,E2 -30419.216} C_VEL
LIN {X 0,Y 171.321,Z 324.196,A -85,B 0,C 180,E1 -30419.401,E2 -30419.401} C_VEL
LIN {X 0,Y 171.372,Z 323.828,A -85,B 0,C 180,E1 -30420,E2 -30420} C_VEL
LIN {X 0,Y 171.309,Z 324.201,A -85,B 0,C 180,E1 -30420.987,E2 -30420.987} C_VEL
LIN {X 0,Y 167.58,Z 339.992,A -85,B 0,C 180,E1 -30421.279,E2 -30421.279} C_VEL
LIN {X 0,Y 164.905,Z 348.529,A -85,B 0,C 180,E1 -30421.5,E2 -30421.5} C_VEL
LIN {X 0,Y 164.798,Z 349.182,A -85,B 0,C 180,E1 -30421.509,E2 -30421.509} C_VEL
LIN {X 0,Y 164.798,Z 406.965,A -85,B 0,C 180,E1 -30421.509,E2 -30421.509} C_VEL
LIN {X 0,Y 146.1,Z 406.965,A -85,B 0,C 180,E1 -30420.567,E2 -30420.567} C_VEL
LIN {X 0,Y 144.121,Z 404.965,A -85,B 0,C 180,E1 -30420.453,E2 -30420.453} C_VEL
LIN {X 0,Y 144.121,Z 396.324,A -85,B 0,C 180,E1 -30420.453,E2 -30420.453} C_VEL
LIN {X 0,Y 140.57,Z 395.115,A -85,B 0,C 180,E1 -30420.674,E2 -30420.674} C_VEL
LIN {X 0,Y 131.146,Z 406.876,A -85,B 0,C 180,E1 -30421.344,E2 -30421.344} C_VEL
LIN {X 0,Y 121.32,Z 417.251,A -85,B 0,C 180,E1 -30422.166,E2 -30422.166} C_VEL
LIN {X 0,Y 109.117,Z 428.037,A -85,B 0,C 180,E1 -30423.315,E2 -30423.315} C_VEL
LIN {X 0,Y 98.728,Z 435.769,A -85,B 0,C 180,E1 -30424.729,E2 -30424.729} C_VEL
LIN {X 0,Y 88.387,Z 442.394,A -85,B 0,C 180,E1 -30426.321,E2 -30426.321} C_VEL
LIN {X 0,Y 74.732,Z 449.716,A -85,B 0,C 180,E1 -30429.089,E2 -30429.089} C_VEL
LIN {X 0,Y 61.292,Z 455.519,A -85,B 0,C 180,E1 -30432.944,E2 -30432.944} C_VEL
LIN {X 0,Y 51.495,Z 458.947,A -85,B 0,C 180,E1 -30437.184,E2 -30437.184} C_VEL
LIN {X 0,Y 39.038,Z 462.409,A -85,B 0,C 180,E1 -30445.823,E2 -30445.823} C_VEL
LIN {X 0,Y 28.184,Z 464.681,A -85,B 0,C 180,E1 -30461.576,E2 -30461.576} C_VEL
LIN {X 0,Y 21.083,Z 465.826,A -85,B 0,C 180,E1 -30490.528,E2 -30490.528} C_VEL
LIN {X 0,Y 20.156,Z 465.975,A -85,B 0,C 180,E1 -30510.001,E2 -30510.001} C_VEL
LIN {X 0,Y 23.909,Z 465.419,A -85,B 0,C 180,E1 -30546.009,E2 -30546.009} C_VEL
LIN {X 0,Y 33.286,Z 463.752,A -85,B 0,C 180,E1 -30567.627,E2 -30567.627} C_VEL
LIN {X 0,Y 45.148,Z 460.923,A -85,B 0,C 180,E1 -30579.069,E2 -30579.069} C_VEL
LIN {X 0,Y 58.548,Z 456.654,A -85,B 0,C 180,E1 -30586.108,E2 -30586.108} C_VEL
LIN {X 0,Y 71.328,Z 451.478,A -85,B 0,C 180,E1 -30590.17,E2 -30590.17} C_VEL
LIN {X 0,Y 84.938,Z 444.605,A -85,B 0,C 180,E1 -30593.176,E2 -30593.176} C_VEL
LIN {X 0,Y 97,Z 437.212,A -85,B 0,C 180,E1 -30595.033,E2 -30595.033} C_VEL
LIN {X 0,Y 107.373,Z 429.65,A -85,B 0,C 180,E1 -30596.543,E2 -30596.543} C_VEL
LIN {X 0,Y 117.824,Z 420.822,A -85,B 0,C 180,E1 -30597.591,E2 -30597.591} C_VEL
LIN {X 0,Y 128.304,Z 410.411,A -85,B 0,C 180,E1 -30598.526,E2 -30598.526} C_VEL
LIN {X 0,Y 137.937,Z 399.077,A -85,B 0,C 180,E1 -30599.247,E2 -30599.247} C_VEL
LIN {X 0,Y 140.568,Z 395.568,A -85,B 0,C 180,E1 -30599.42,E2 -30599.42} C_VEL
LIN {X 0,Y 140.565,Z 395.58,A -85,B 0,C 180,E1 -30599.588,E2 -30599.588} C_VEL
LIN {X 0,Y 130.777,Z 407.722,A -85,B 0,C 180,E1 -30600.205,E2 -30600.205} C_VEL
LIN {X 0,Y 121.248,Z 417.757,A -85,B 0,C 180,E1 -30600.881,E2 -30600.881} C_VEL
LIN {X 0,Y 110.743,Z 427.146,A -85,B 0,C 180,E1 -30601.74,E2 -30601.74} C_VEL
LIN {X 0,Y 98.531,Z 436.385,A -85,B 0,C 180,E1 -30603.031,E2 -30603.031} C_VEL
LIN {X 0,Y 84.676,Z 445.095,A -85,B 0,C 180,E1 -30605.13,E2 -30605.13} C_VEL
LIN {X 0,Y 70.973,Z 452.092,A -85,B 0,C 180,E1 -30608.009,E2 -30608.009} C_VEL
LIN {X 0,Y 57.511,Z 457.598,A -85,B 0,C 180,E1 -30612.141,E2 -30612.141} C_VEL
LIN {X 0,Y 44.543,Z 461.773,A -85,B 0,C 180,E1 -30618.794,E2 -30618.794} C_VEL
